C01874=87.153,47.905,41.515,178.9994,1.0610,0.0000
C01875=89.570,44.326,41.678,179.9701,0.0579,0.0000
C01876=91.502,40.323,41.785,179.9964,0.0081,0.0000
C01877=93.214,36.189,41.785,179.9968,0.0083,0.0000
C01878=94.679,31.992,41.678,179.9802,0.0621,0.0000
C01879=95.500,27.752,41.515,179.9573,1.4576,0.0000
C01880=94.968,23.775,41.355,-179.3183,2.1553,0.0000
C01881=93.250,20.743,41.159,-177.2598,2.8295,0.0000
C01882=90.644,19.021,40.789,-176.5682,1.8279,0.0000
C01883=87.735,17.640,40.048,-179.2135,0.3689,0.0000
C01884=85.134,16.299,39.090,175.2426,-2.7030,0.0000
C01885=83.232,14.718,38.165,166.7718,-12.7923,0.0000
C01886=82.260,12.305,37.495,171.8942,-33.8546,0.0000
C01887=82.270,8.324,37.229,-177.9072,-37.5897,0.0000
C01888=82.553,4.208,37.217,-177.5804,-37.7646,0.0000
C01889=82.662,0.000,37.225,179.9996,-37.7945,0.0000
C01890=82.553,-4.208,37.217,177.5810,-37.7647,0.0000
C01891=82.270,-8.324,37.229,177.9089,-37.5895,0.0000
C01892=82.260,-12.305,37.495,-171.8950,-33.8549,0.0000
C01893=83.232,-14.718,38.165,-166.7718,-12.7923,0.0000
C01894=85.134,-16.299,39.090,-175.2426,-2.7030,0.0000
C01895=87.735,-17.640,40.048,179.2135,0.3689,0.0000
C01896=90.644,-19.021,40.789,176.5682,1.8279,0.0000
C01897=93.250,-20.743,41.159,177.2598,2.8295,0.0000
C01898=94.968,-23.775,41.355,179.3183,2.1553,0.0000
C01899=95.500,-27.752,41.515,-179.9573,1.4576,0.0000
C01900=94.679,-31.992,41.678,-179.9802,0.0621,0.0000
C01901=93.214,-36.189,41.785,-179.9968,0.0083,0.0000
C01902=91.502,-40.323,41.785,-179.9964,0.0081,0.0000
C01903=89.570,-44.326,41.678,-179.9701,0.0579,0.0000
C01904=87.153,-47.905,41.515,-178.9994,1.0610,0.0000
C01905=83.964,-50.341,41.355,-177.9940,1.0426,0.0000
C01906=80.606,-51.270,41.159,-176.0647,0.0633,0.0000
C01907=77.545,-50.645,40.789,-176.2827,-1.1365,0.0000
C01908=74.511,-49.565,40.048,-179.1830,-0.2954,0.0000
C01909=71.724,-48.673,39.090,174.7304,1.4587,0.0000
C01910=69.261,-48.447,38.165,161.9042,0.3246,0.0000
C01911=66.868,-49.465,37.495,150.0988,-20.4873,0.0000
C01912=64.059,-52.288,37.229,152.5931,-29.6910,0.0000
C01913=61.349,-55.398,37.217,152.6199,-30.0136,0.0000
C01914=58.451,-58.451,37.225,151.2604,-28.7392,0.0000
C01915=55.398,-61.349,37.217,149.9866,-27.3805,0.0000
C01916=52.288,-64.059,37.229,150.3100,-27.4077,0.0000
C01917=49.465,-66.868,37.495,159.5118,-29.9009,0.0000
C01918=48.447,-69.261,38.165,-179.6754,-18.0958,0.0000
C01919=48.673,-71.724,39.090,-178.5413,-5.2696,0.0000
C01920=49.565,-74.511,40.048,179.7046,0.8170,0.0000
C01921=50.645,-77.545,40.789,178.8635,3.7173,0.0000
C01922=51.270,-80.606,41.159,-179.9367,3.9353,0.0000
C01923=50.341,-83.964,41.355,-178.9574,2.0060,0.0000
C01924=47.905,-87.153,41.515,-178.9390,1.0006,0.0000
C01925=44.326,-89.570,41.678,-179.9421,0.0299,0.0000
C01926=40.323,-91.502,41.785,-179.9919,0.0036,0.0000
C01927=36.189,-93.214,41.785,-179.9917,0.0032,0.0000
C01928=31.992,-94.679,41.678,-179.9379,0.0198,0.0000
C01929=27.752,-95.500,41.515,-178.5424,0.0427,0.0000
C01930=23.775,-94.968,41.355,-177.8447,-0.6817,0.0000
C01931=20.743,-93.250,41.159,-177.1705,-2.7402,0.0000
C01932=19.021,-90.644,40.789,-178.1721,-3.4318,0.0000
C01933=17.640,-87.735,40.048,-179.6311,-0.7865,0.0000
C01934=16.299,-85.134,39.090,177.2970,4.7574,0.0000
C01935=14.718,-83.232,38.165,167.2077,13.2282,0.0000
C01936=12.305,-82.260,37.495,146.1454,8.1058,0.0000
C01937=8.324,-82.270,37.229,142.4103,-2.0928,0.0000
C01938=4.208,-82.553,37.217,142.2354,-2.4196,0.0000
C01939=0.000,-82.662,37.225,142.2055,0.0004,0.0000
C01940=0.000,-82.662,37.225,142.2055,0.0004,0.0000
C01941=-4.208,-82.553,37.217,142.2353,2.4190,0.0000
C01942=-8.324,-82.270,37.229,142.4105,2.0911,0.0000
C01943=-12.305,-82.260,37.495,146.1451,-8.1050,0.0000
C01944=-14.718,-83.232,38.165,167.2077,-13.2282,0.0000
C01945=-16.299,-85.134,39.090,177.2970,-4.7574,0.0000
C01946=-17.640,-87.735,40.048,-179.6311,0.7865,0.0000
C01947=-19.021,-90.644,40.789,-178.1721,3.4318,0.0000
C01948=-20.743,-93.250,41.159,-177.1705,2.7402,0.0000
C01949=-23.775,-94.968,41.355,-177.8447,0.6817,0.0000
C01950=-27.752,-95.500,41.515,-178.5424,-0.0427,0.0000
C01951=-31.992,-94.679,41.678,-179.9379,-0.0198,0.0000
C01952=-36.189,-93.214,41.785,-179.9917,-0.0032,0.0000
C01953=-40.323,-91.502,41.785,-179.9919,-0.0036,0.0000
C01954=-44.326,-89.570,41.678,-179.9421,-0.0299,0.0000
C01955=-47.905,-87.153,41.515,-178.9390,-1.0006,0.0000
C01956=-50.341,-83.964,41.355,-178.9574,-2.0060,0.0000
C01957=-51.270,-80.606,41.159,-179.9367,-3.9353,0.0000
C01958=-50.645,-77.545,40.789,178.8635,-3.7173,0.0000
C01959=-49.565,-74.511,40.048,179.7046,-0.8170,0.0000
C01960=-48.673,-71.724,39.090,-178.5413,5.2696,0.0000
C01961=-48.447,-69.261,38.165,-179.6754,18.0958,0.0000
C01962=-49.465,-66.868,37.495,159.5127,29.9012,0.0000
C01963=-52.288,-64.059,37.229,150.3090,27.4069,0.0000
C01964=-55.398,-61.349,37.217,149.9864,27.3801,0.0000
C01965=-58.451,-58.451,37.225,151.2608,28.7396,0.0000
C01966=-61.349,-55.398,37.217,152.6195,30.0134,0.0000
C01967=-64.059,-52.288,37.229,152.5923,29.6900,0.0000
C01968=-66.868,-49.465,37.495,150.0991,20.4882,0.0000
C01969=-69.261,-48.447,38.165,161.9042,-0.3246,0.0000
C01970=-71.724,-48.673,39.090,174.7304,-1.4587,0.0000
C01971=-74.511,-49.565,40.048,-179.1830,0.2954,0.0000
C01972=-77.545,-50.645,40.789,-176.2827,1.1365,0.0000
C01973=-80.606,-51.270,41.159,-176.0647,-0.0633,0.0000
C01974=-83.964,-50.341,41.355,-177.9940,-1.0426,0.0000
C01975=-87.153,-47.905,41.515,-178.9994,-1.0610,0.0000
C01976=-89.570,-44.326,41.678,-179.9701,-0.0579,0.0000
C01977=-91.502,-40.323,41.785,-179.9964,-0.0081,0.0000
C01978=-93.214,-36.189,41.785,-179.9968,-0.0083,0.0000
C01979=-94.679,-31.992,41.678,-179.9802,-0.0621,0.0000
C01980=-95.500,-27.752,41.515,-179.9573,-1.4576,0.0000
C01981=-94.968,-23.775,41.355,179.3183,-2.1553,0.0000
C01982=-93.250,-20.743,41.159,177.2598,-2.8295,0.0000
C01983=-90.644,-19.021,40.789,176.5682,-1.8279,0.0000
C01984=-87.735,-17.640,40.048,179.2135,-0.3689,0.0000
C01985=-85.134,-16.299,39.090,-175.2426,2.7030,0.0000
C01986=-83.232,-14.718,38.165,-166.7718,12.7923,0.0000
C01987=-82.260,-12.305,37.495,-171.8942,33.8546,0.0000
C01988=-82.270,-8.324,37.229,177.9072,37.5897,0.0000
C01989=-82.553,-4.208,37.217,177.5804,37.7646,0.0000
C01990=-82.662,0.000,37.225,-179.9996,37.7945,0.0000
C01991=-82.553,4.208,37.217,-177.5810,37.7647,0.0000
C01992=-82.270,8.324,37.229,-177.9089,37.5895,0.0000
C01993=-82.260,12.305,37.495,171.8950,33.8549,0.0000
C01994=-83.232,14.718,38.165,166.7718,12.7923,0.0000
C01995=-85.134,16.299,39.090,175.2426,2.7030,0.0000
C01996=-87.735,17.640,40.048,-179.2135,-0.3689,0.0000
C01997=-90.644,19.021,40.789,-176.5682,-1.8279,0.0000
C01998=-93.250,20.743,41.159,-177.2598,-2.8295,0.0000
C01999=-94.968,23.775,41.355,-179.3183,-2.1553,0.0000
///TOOL 0
///POSTYPE ANGLE
///ANGLE
EC00000=-33.2751,0.0000
EC00001=-32.3830,0.0000
EC00002=-31.4965,0.0000
EC00003=-30.3670,0.0000
EC00004=-28.7935,0.0000
EC00005=-26.9678,0.0000
EC00006=-25.1253,0.0000
EC00007=-23.3660,0.0000
EC00008=-21.6343,0.0000
EC00009=-19.8748,0.0000
EC00010=-18.0324,0.0000
EC00011=-16.2063,0.0000
EC00012=-14.6333,0.0000
EC00013=-13.5035,0.0000
EC00014=-12.6169,0.0000
EC00015=-11.7253,0.0000
EC00016=-10.5819,0.0000
EC00017=-8.8371,0.0000
EC00018=-6.1699,0.0000
EC00019=-3.2152,0.0000
EC00020=0.0000,0.0000
EC00021=0.0000,0.0000
EC00022=3.1930,0.0000
EC00023=6.1402,0.0000
EC00024=8.8129,0.0000
EC00025=10.5402,0.0000
EC00026=11.6582,0.0000
EC00027=12.5225,0.0000
EC00028=13.3766,0.0000
EC00029=14.4702,0.0000
EC00030=16.0363,0.0000
EC00031=17.8866,0.0000
EC00032=19.7782,0.0000
EC00033=21.6011,0.0000
EC00034=23.3991,0.0000
EC00035=25.2213,0.0000
EC00036=27.1138,0.0000
EC00037=28.9637,0.0000
EC00038=30.5297,0.0000
EC00039=31.6234,0.0000
EC00040=32.4779,0.0000
EC00041=33.3415,0.0000
EC00042=34.4600,0.0000
EC00043=36.1873,0.0000
EC00044=38.8598,0.0000
EC00045=41.8071,0.0000
EC00046=45.0000,0.0000
EC00047=48.1929,0.0000
EC00048=51.1402,0.0000
EC00049=53.8127,0.0000
EC00050=55.5400,0.0000
EC00051=56.6585,0.0000
EC00052=57.5221,0.0000
EC00053=58.3766,0.0000
EC00054=59.4703,0.0000
EC00055=61.0363,0.0000
EC00056=62.8862,0.0000
EC00057=64.7787,0.0000
EC00058=66.6009,0.0000
EC00059=68.3989,0.0000
EC00060=70.2218,0.0000
EC00061=72.1134,0.0000
EC00062=73.9637,0.0000
EC00063=75.5298,0.0000
EC00064=76.6234,0.0000
EC00065=77.4775,0.0000
EC00066=78.3418,0.0000
EC00067=79.4598,0.0000
EC00068=81.1871,0.0000
EC00069=83.8598,0.0000
EC00070=86.8070,0.0000
EC00071=90.0000,0.0000
EC00072=93.1930,0.0000
EC00073=96.1402,0.0000
EC00074=98.8128,0.0000
EC00075=100.5402,0.0000
EC00076=101.6582,0.0000
EC00077=102.5225,0.0000
EC00078=103.3766,0.0000
EC00079=104.4702,0.0000
EC00080=106.0363,0.0000
EC00081=107.8866,0.0000
EC00082=109.7782,0.0000
EC00083=111.6011,0.0000
EC00084=113.3991,0.0000
EC00085=115.2213,0.0000
EC00086=117.1138,0.0000
EC00087=118.9637,0.0000
EC00088=120.5297,0.0000
EC00089=121.6234,0.0000
EC00090=122.4779,0.0000
EC00091=123.3415,0.0000
EC00092=124.4600,0.0000
EC00093=126.1873,0.0000
EC00094=128.8598,0.0000
EC00095=131.8071,0.0000
EC00096=135.0000,0.0000
EC00097=138.1929,0.0000
EC00098=141.1402,0.0000
EC00099=143.8127,0.0000
EC00100=145.5400,0.0000
EC00101=146.6585,0.0000
EC00102=147.5221,0.0000
EC00103=148.3766,0.0000
EC00104=149.4703,0.0000
EC00105=151.0363,0.0000
EC00106=152.8862,0.0000
EC00107=154.7787,0.0000
EC00108=156.6009,0.0000
EC00109=158.3989,0.0000
EC00110=160.2218,0.0000
EC00111=162.1134,0.0000
EC00112=163.9637,0.0000
EC00113=165.5298,0.0000
EC00114=166.6234,0.0000
EC00115=167.4775,0.0000
EC00116=168.3418,0.0000
EC00117=169.4598,0.0000
EC00118=171.1871,0.0000
EC00119=173.8598,0.0000
EC00120=176.8070,0.0000
EC00121=180.0000,0.0000
EC00122=180.0000,0.0000
EC00123=-176.8070,0.0000
EC00124=-173.8598,0.0000
EC00125=-171.1872,0.0000
EC00126=-169.4598,0.0000
EC00127=-168.3418,0.0000
EC00128=-167.4775,0.0000
EC00129=-166.6234,0.0000
EC00130=-165.5298,0.0000
EC00131=-163.9637,0.0000
EC00132=-162.1134,0.0000
EC00133=-160.2218,0.0000
EC00134=-158.3989,0.0000
EC00135=-156.6009,0.0000
EC00136=-154.7787,0.0000
EC00137=-152.8862,0.0000
EC00138=-151.0363,0.0000
EC00139=-149.4703,0.0000
EC00140=-148.3766,0.0000
EC00141=-147.5221,0.0000
EC00142=-146.6585,0.0000
EC00143=-145.5400,0.0000
EC00144=-143.8127,0.0000
EC00145=-141.1402,0.0000
EC00146=-138.1929,0.0000
EC00147=-135.0000,0.0000
EC00148=-131.8071,0.0000
EC00149=-128.8598,0.0000
EC00150=-126.1873,0.0000
EC00151=-124.4600,0.0000
EC00152=-123.3415,0.0000
EC00153=-122.4779,0.0000
EC00154=-121.6234,0.0000
EC00155=-120.5297,0.0000
EC00156=-118.9637,0.0000
EC00157=-117.1138,0.0000
EC00158=-115.2213,0.0000
EC00159=-113.3991,0.0000
EC00160=-111.6011,0.0000
EC00161=-109.7782,0.0000
EC00162=-107.8866,0.0000
EC00163=-106.0363,0.0000
EC00164=-104.4702,0.0000
EC00165=-103.3766,0.0000
EC00166=-102.5225,0.0000
EC00167=-101.6582,0.0000
EC00168=-100.5402,0.0000
EC00169=-98.8129,0.0000
EC00170=-96.1402,0.0000
EC00171=-93.1930,0.0000
EC00172=-90.0000,0.0000
EC00173=-86.8070,0.0000
EC00174=-83.8598,0.0000
EC00175=-81.1872,0.0000
EC00176=-79.4598,0.0000
EC00177=-78.3418,0.0000
EC00178=-77.4775,0.0000
EC00179=-76.6234,0.0000
EC00180=-75.5298,0.0000
EC00181=-73.9637,0.0000
EC00182=-72.1134,0.0000
EC00183=-70.2218,0.0000
EC00184=-68.3989,0.0000
EC00185=-66.6009,0.0000
EC00186=-64.7787,0.0000
EC00187=-62.8862,0.0000
EC00188=-61.0363,0.0000
EC00189=-59.4703,0.0000
EC00190=-58.3766,0.0000
EC00191=-57.5221,0.0000
EC00192=-56.6585,0.0000
EC00193=-55.5400,0.0000
EC00194=-53.8127,0.0000
EC00195=-51.1402,0.0000
EC00196=-48.1929,0.0000
EC00197=-45.0000,0.0000
EC00198=-41.8071,0.0000
EC00199=-38.8598,0.0000
EC00200=-36.1873,0.0000
EC00201=-34.4600,0.0000
EC00202=-33.3415,0.0000
EC00203=-32.4779,0.0000
EC00204=-31.6234,0.0000
EC00205=-30.5297,0.0000
EC00206=-28.9637,0.0000
EC00207=-27.1138,0.0000
EC00208=-25.2213,0.0000
EC00209=-23.3991,0.0000
EC00210=-21.6011,0.0000
EC00211=-19.7782,0.0000
EC00212=-17.8866,0.0000
EC00213=-16.0363,0.0000
EC00214=-14.4702,0.0000
EC00215=-13.3766,0.0000
EC00216=-12.5225,0.0000
EC00217=-11.6582,0.0000
EC00218=-10.5402,0.0000
EC00219=-8.8128,0.0000
EC00220=-6.1402,0.0000
EC00221=-3.1930,0.0000
EC00222=0.0000,0.0000
EC00223=0.0000,0.0000
EC00224=3.1693,0.0000
EC00225=6.1086,0.0000
EC00226=8.7858,0.0000
EC00227=10.4951,0.0000
EC00228=11.5862,0.0000
EC00229=12.4199,0.0000
EC00230=13.2394,0.0000
EC00231=14.2944,0.0000
EC00232=15.8535,0.0000
EC00233=17.7299,0.0000
EC00234=19.6757,0.0000
EC00235=21.5655,0.0000
EC00236=23.4348,0.0000
EC00237=25.3246,0.0000
EC00238=27.2701,0.0000
EC00239=29.1464,0.0000
EC00240=30.7059,0.0000
EC00241=31.7605,0.0000
EC00242=32.5800,0.0000
EC00243=33.4139,0.0000
EC00244=34.5045,0.0000
EC00245=36.2144,0.0000
EC00246=38.8913,0.0000
EC00247=41.8309,0.0000
EC00248=45.0000,0.0000
EC00249=48.1691,0.0000
EC00250=51.1087,0.0000
EC00251=53.7856,0.0000
EC00252=55.4955,0.0000
EC00253=56.5861,0.0000
EC00254=57.4200,0.0000
EC00255=58.2395,0.0000
EC00256=59.2941,0.0000
EC00257=60.8536,0.0000
EC00258=62.7299,0.0000
EC00259=64.6754,0.0000
EC00260=66.5652,0.0000
EC00261=68.4345,0.0000
EC00262=70.3243,0.0000
EC00263=72.2701,0.0000
EC00264=74.1465,0.0000
EC00265=75.7056,0.0000
EC00266=76.7606,0.0000
EC00267=77.5801,0.0000
EC00268=78.4138,0.0000
EC00269=79.5049,0.0000
EC00270=81.2142,0.0000
EC00271=83.8914,0.0000
EC00272=86.8307,0.0000
EC00273=90.0000,0.0000
EC00274=93.1693,0.0000
EC00275=96.1086,0.0000
EC00276=98.7858,0.0000
EC00277=100.4951,0.0000
EC00278=101.5862,0.0000
EC00279=102.4199,0.0000
EC00280=103.2394,0.0000
EC00281=104.2944,0.0000
EC00282=105.8535,0.0000
EC00283=107.7299,0.0000
EC00284=109.6757,0.0000
EC00285=111.5655,0.0000
EC00286=113.4348,0.0000
EC00287=115.3246,0.0000
EC00288=117.2701,0.0000
EC00289=119.1464,0.0000
EC00290=120.7059,0.0000
EC00291=121.7605,0.0000
EC00292=122.5800,0.0000
EC00293=123.4139,0.0000
EC00294=124.5045,0.0000
EC00295=126.2144,0.0000
EC00296=128.8913,0.0000
EC00297=131.8309,0.0000
EC00298=135.0000,0.0000
EC00299=138.1691,0.0000
EC00300=141.1087,0.0000
EC00301=143.7856,0.0000
EC00302=145.4955,0.0000
EC00303=146.5861,0.0000
EC00304=147.4200,0.0000
EC00305=148.2395,0.0000
EC00306=149.2941,0.0000
EC00307=150.8536,0.0000
EC00308=152.7299,0.0000
EC00309=154.6754,0.0000
EC00310=156.5652,0.0000
EC00311=158.4345,0.0000
EC00312=160.3243,0.0000
EC00313=162.2701,0.0000
EC00314=164.1465,0.0000
EC00315=165.7056,0.0000
EC00316=166.7606,0.0000
EC00317=167.5801,0.0000
EC00318=168.4138,0.0000
EC00319=169.5049,0.0000
EC00320=171.2142,0.0000
EC00321=173.8914,0.0000
EC00322=176.8307,0.0000
EC00323=180.0000,0.0000
EC00324=180.0000,0.0000
EC00325=-176.8307,0.0000
EC00326=-173.8914,0.0000
EC00327=-171.2142,0.0000
EC00328=-169.5049,0.0000
EC00329=-168.4138,0.0000
EC00330=-167.5801,0.0000
EC00331=-166.7606,0.0000
EC00332=-165.7056,0.0000
EC00333=-164.1465,0.0000
EC00334=-162.2701,0.0000
EC00335=-160.3243,0.0000
EC00336=-158.4345,0.0000
EC00337=-156.5652,0.0000
EC00338=-154.6754,0.0000
EC00339=-152.7299,0.0000
EC00340=-150.8536,0.0000
EC00341=-149.2941,0.0000
EC00342=-148.2395,0.0000
EC00343=-147.4200,0.0000
EC00344=-146.5861,0.0000
EC00345=-145.4955,0.0000
EC00346=-143.7856,0.0000
EC00347=-141.1087,0.0000
EC00348=-138.1691,0.0000
EC00349=-135.0000,0.0000
EC00350=-131.8309,0.0000
EC00351=-128.8913,0.0000
EC00352=-126.2144,0.0000
EC00353=-124.5045,0.0000
EC00354=-123.4139,0.0000
EC00355=-122.5800,0.0000
EC00356=-121.7605,0.0000
EC00357=-120.7059,0.0000
EC00358=-119.1464,0.0000
EC00359=-117.2701,0.0000
EC00360=-115.3246,0.0000
EC00361=-113.4348,0.0000
EC00362=-111.5655,0.0000
EC00363=-109.6757,0.0000
EC00364=-107.7299,0.0000
EC00365=-105.8535,0.0000
EC00366=-104.2944,0.0000
EC00367=-103.2394,0.0000
EC00368=-102.4199,0.0000
EC00369=-101.5862,0.0000
EC00370=-100.4951,0.0000
EC00371=-98.7858,0.0000
EC00372=-96.1086,0.0000
EC00373=-93.1693,0.0000
EC00374=-90.0000,0.0000
EC00375=-86.8307,0.0000
EC00376=-83.8914,0.0000
EC00377=-81.2142,0.0000
EC00378=-79.5049,0.0000
EC00379=-78.4138,0.0000
EC00380=-77.5801,0.0000
EC00381=-76.7606,0.0000
EC00382=-75.7056,0.0000
EC00383=-74.1465,0.0000
EC00384=-72.2701,0.0000
EC00385=-70.3243,0.0000
EC00386=-68.4345,0.0000
EC00387=-66.5652,0.0000
EC00388=-64.6754,0.0000
EC00389=-62.7299,0.0000
EC00390=-60.8536,0.0000
EC00391=-59.2941,0.0000
EC00392=-58.2395,0.0000
EC00393=-57.4200,0.0000
EC00394=-56.5861,0.0000
EC00395=-55.4955,0.0000
EC00396=-53.7856,0.0000
EC00397=-51.1087,0.0000
EC00398=-48.1691,0.0000
EC00399=-45.0000,0.0000
EC00400=-41.8309,0.0000
EC00401=-38.8913,0.0000
EC00402=-36.2144,0.0000
EC00403=-34.5045,0.0000
EC00404=-33.4139,0.0000
EC00405=-32.5800,0.0000
EC00406=-31.7605,0.0000
EC00407=-30.7059,0.0000
EC00408=-29.1464,0.0000
EC00409=-27.2701,0.0000
EC00410=-25.3246,0.0000
EC00411=-23.4348,0.0000
EC00412=-21.5655,0.0000
EC00413=-19.6757,0.0000
EC00414=-17.7299,0.0000
EC00415=-15.8535,0.0000
EC00416=-14.2944,0.0000
EC00417=-13.2394,0.0000
EC00418=-12.4199,0.0000
EC00419=-11.5862,0.0000
EC00420=-10.4951,0.0000
EC00421=-8.7858,0.0000
EC00422=-6.1086,0.0000
EC00423=-3.1693,0.0000
EC00424=0.0000,0.0000
EC00425=0.0000,0.0000
EC00426=3.1434,0.0000
EC00427=6.0750,0.0000
EC00428=8.7577,0.0000
EC00429=10.4474,0.0000
EC00430=11.5089,0.0000
EC00431=12.3101,0.0000
EC00432=13.0930,0.0000
EC00433=14.1066,0.0000
EC00434=15.6587,0.0000
EC00435=17.5637,0.0000
EC00436=19.5659,0.0000
EC00437=21.5274,0.0000
EC00438=23.4725,0.0000
EC00439=25.4343,0.0000
EC00440=27.4359,0.0000
EC00441=29.3411,0.0000
EC00442=30.8935,0.0000
EC00443=31.9071,0.0000
EC00444=32.6899,0.0000
EC00445=33.4910,0.0000
EC00446=34.5530,0.0000
EC00447=36.2423,0.0000
EC00448=38.9252,0.0000
EC00449=41.8567,0.0000
EC00450=45.0000,0.0000
EC00451=48.1433,0.0000
EC00452=51.0748,0.0000
EC00453=53.7577,0.0000
EC00454=55.4470,0.0000
EC00455=56.5090,0.0000
EC00456=57.3101,0.0000
EC00457=58.0929,0.0000
EC00458=59.1065,0.0000
EC00459=60.6589,0.0000
EC00460=62.5641,0.0000
EC00461=64.5657,0.0000
EC00462=66.5275,0.0000
EC00463=68.4726,0.0000
EC00464=70.4341,0.0000
EC00465=72.4363,0.0000
EC00466=74.3413,0.0000
EC00467=75.8934,0.0000
EC00468=76.9070,0.0000
EC00469=77.6899,0.0000
EC00470=78.4911,0.0000
EC00471=79.5526,0.0000
EC00472=81.2423,0.0000
EC00473=83.9250,0.0000
EC00474=86.8566,0.0000
EC00475=90.0000,0.0000
EC00476=93.1434,0.0000
EC00477=96.0750,0.0000
EC00478=98.7577,0.0000
EC00479=100.4474,0.0000
EC00480=101.5089,0.0000
EC00481=102.3101,0.0000
EC00482=103.0930,0.0000
EC00483=104.1066,0.0000
EC00484=105.6587,0.0000
EC00485=107.5637,0.0000
EC00486=109.5659,0.0000
EC00487=111.5274,0.0000
EC00488=113.4725,0.0000
EC00489=115.4343,0.0000
EC00490=117.4359,0.0000
EC00491=119.3411,0.0000
EC00492=120.8935,0.0000
EC00493=121.9071,0.0000
EC00494=122.6899,0.0000
EC00495=123.4910,0.0000
EC00496=124.5530,0.0000
EC00497=126.2423,0.0000
EC00498=128.9252,0.0000
EC00499=131.8567,0.0000
EC00500=135.0000,0.0000
EC00501=138.1433,0.0000
EC00502=141.0748,0.0000
EC00503=143.7577,0.0000
EC00504=145.4470,0.0000
EC00505=146.5090,0.0000
EC00506=147.3101,0.0000
EC00507=148.0929,0.0000
EC00508=149.1065,0.0000
EC00509=150.6589,0.0000
EC00510=152.5641,0.0000
EC00511=154.5657,0.0000
EC00512=156.5275,0.0000
EC00513=158.4726,0.0000
EC00514=160.4341,0.0000
EC00515=162.4363,0.0000
EC00516=164.3413,0.0000
EC00517=165.8934,0.0000
EC00518=166.9070,0.0000
EC00519=167.6899,0.0000
EC00520=168.4911,0.0000
EC00521=169.5526,0.0000
EC00522=171.2423,0.0000
EC00523=173.9250,0.0000
EC00524=176.8566,0.0000
EC00525=180.0000,0.0000
EC00526=180.0000,0.0000
EC00527=-176.8566,0.0000
EC00528=-173.9250,0.0000
EC00529=-171.2423,0.0000
EC00530=-169.5526,0.0000
EC00531=-168.4911,0.0000
EC00532=-167.6899,0.0000
EC00533=-166.9070,0.0000
EC00534=-165.8934,0.0000
EC00535=-164.3413,0.0000
EC00536=-162.4363,0.0000
EC00537=-160.4341,0.0000
EC00538=-158.4726,0.0000
EC00539=-156.5275,0.0000
EC00540=-154.5657,0.0000
EC00541=-152.5641,0.0000
EC00542=-150.6589,0.0000
EC00543=-149.1065,0.0000
EC00544=-148.0929,0.0000
EC00545=-147.3101,0.0000
EC00546=-146.5090,0.0000
EC00547=-145.4470,0.0000
EC00548=-143.7577,0.0000
EC00549=-141.0748,0.0000
EC00550=-138.1433,0.0000
EC00551=-135.0000,0.0000
EC00552=-131.8567,0.0000
EC00553=-128.9252,0.0000
EC00554=-126.2423,0.0000
EC00555=-124.5530,0.0000
EC00556=-123.4910,0.0000
EC00557=-122.6899,0.0000
EC00558=-121.9071,0.0000
EC00559=-120.8935,0.0000
EC00560=-119.3411,0.0000
EC00561=-117.4359,0.0000
EC00562=-115.4343,0.0000
EC00563=-113.4725,0.0000
EC00564=-111.5274,0.0000
EC00565=-109.5659,0.0000
EC00566=-107.5637,0.0000
EC00567=-105.6587,0.0000
EC00568=-104.1066,0.0000
EC00569=-103.0930,0.0000
EC00570=-102.3101,0.0000
EC00571=-101.5089,0.0000
EC00572=-100.4474,0.0000
EC00573=-98.7577,0.0000
EC00574=-96.0750,0.0000
EC00575=-93.1434,0.0000
EC00576=-90.0000,0.0000
EC00577=-86.8566,0.0000
EC00578=-83.9250,0.0000
EC00579=-81.2423,0.0000
EC00580=-79.5526,0.0000
EC00581=-78.4911,0.0000
EC00582=-77.6899,0.0000
EC00583=-76.9070,0.0000
EC00584=-75.8934,0.0000
EC00585=-74.3413,0.0000
EC00586=-72.4363,0.0000
EC00587=-70.4341,0.0000
EC00588=-68.4726,0.0000
EC00589=-66.5275,0.0000
EC00590=-64.5657,0.0000
EC00591=-62.5641,0.0000
EC00592=-60.6589,0.0000
EC00593=-59.1065,0.0000
EC00594=-58.0929,0.0000
EC00595=-57.3101,0.0000
EC00596=-56.5090,0.0000
EC00597=-55.4470,0.0000
EC00598=-53.7577,0.0000
EC00599=-51.0748,0.0000
EC00600=-48.1433,0.0000
EC00601=-45.0000,0.0000
EC00602=-41.8567,0.0000
EC00603=-38.9252,0.0000
EC00604=-36.2423,0.0000
EC00605=-34.5530,0.0000
EC00606=-33.4910,0.0000
EC00607=-32.6899,0.0000
EC00608=-31.9071,0.0000
EC00609=-30.8935,0.0000
EC00610=-29.3411,0.0000
EC00611=-27.4359,0.0000
EC00612=-25.4343,0.0000
EC00613=-23.4725,0.0000
EC00614=-21.5274,0.0000
EC00615=-19.5659,0.0000
EC00616=-17.5637,0.0000
EC00617=-15.6587,0.0000
EC00618=-14.1066,0.0000
EC00619=-13.0930,0.0000
EC00620=-12.3101,0.0000
EC00621=-11.5089,0.0000
EC00622=-10.4474,0.0000
EC00623=-8.7577,0.0000
EC00624=-6.0750,0.0000
EC00625=-3.1434,0.0000
EC00626=0.0000,0.0000
EC00627=0.0000,0.0000
EC00628=3.1159,0.0000
EC00629=6.0385,0.0000
EC00630=8.7274,0.0000
EC00631=10.3963,0.0000
EC00632=11.4267,0.0000
EC00633=12.1938,0.0000
EC00634=12.9380,0.0000
EC00635=13.9087,0.0000
EC00636=15.4538,0.0000
EC00637=17.3887,0.0000
EC00638=19.4506,0.0000
EC00639=21.4875,0.0000
EC00640=23.5125,0.0000
EC00641=25.5494,0.0000
EC00642=27.6113,0.0000
EC00643=29.5463,0.0000
EC00644=31.0916,0.0000
EC00645=32.0621,0.0000
EC00646=32.8061,0.0000
EC00647=33.5730,0.0000
EC00648=34.6038,0.0000
EC00649=36.2732,0.0000
EC00650=38.9613,0.0000
EC00651=41.8843,0.0000
EC00652=45.0000,0.0000
EC00653=48.1157,0.0000
EC00654=51.0387,0.0000
EC00655=53.7268,0.0000
EC00656=55.3962,0.0000
EC00657=56.4270,0.0000
EC00658=57.1939,0.0000
EC00659=57.9379,0.0000
EC00660=58.9084,0.0000
EC00661=60.4537,0.0000
EC00662=62.3887,0.0000
EC00663=64.4506,0.0000
EC00664=66.4875,0.0000
EC00665=68.5125,0.0000
EC00666=70.5494,0.0000
EC00667=72.6113,0.0000
EC00668=74.5462,0.0000
EC00669=76.0913,0.0000
EC00670=77.0620,0.0000
EC00671=77.8062,0.0000
EC00672=78.5733,0.0000
EC00673=79.6037,0.0000
EC00674=81.2726,0.0000
EC00675=83.9615,0.0000
EC00676=86.8841,0.0000
EC00677=90.0000,0.0000
EC00678=93.1159,0.0000
EC00679=96.0385,0.0000
EC00680=98.7274,0.0000
EC00681=100.3963,0.0000
EC00682=101.4267,0.0000
EC00683=102.1938,0.0000
EC00684=102.9380,0.0000
EC00685=103.9087,0.0000
EC00686=105.4538,0.0000
EC00687=107.3887,0.0000
EC00688=109.4506,0.0000
EC00689=111.4875,0.0000
EC00690=113.5125,0.0000
EC00691=115.5494,0.0000
EC00692=117.6113,0.0000
EC00693=119.5463,0.0000
EC00694=121.0916,0.0000
EC00695=122.0621,0.0000
EC00696=122.8061,0.0000
EC00697=123.5730,0.0000
EC00698=124.6038,0.0000
EC00699=126.2732,0.0000
EC00700=128.9613,0.0000
EC00701=131.8843,0.0000
EC00702=135.0000,0.0000
EC00703=138.1157,0.0000
EC00704=141.0387,0.0000
EC00705=143.7268,0.0000
EC00706=145.3962,0.0000
EC00707=146.4270,0.0000
EC00708=147.1939,0.0000
EC00709=147.9379,0.0000
EC00710=148.9084,0.0000
EC00711=150.4537,0.0000
EC00712=152.3887,0.0000
EC00713=154.4506,0.0000
EC00714=156.4875,0.0000
EC00715=158.5125,0.0000
EC00716=160.5494,0.0000
EC00717=162.6113,0.0000
EC00718=164.5462,0.0000
EC00719=166.0913,0.0000
EC00720=167.0620,0.0000
EC00721=167.8062,0.0000
EC00722=168.5733,0.0000
EC00723=169.6037,0.0000
EC00724=171.2726,0.0000
EC00725=173.9615,0.0000
EC00726=176.8841,0.0000
EC00727=180.0000,0.0000
EC00728=180.0000,0.0000
EC00729=-176.8841,0.0000
EC00730=-173.9615,0.0000
EC00731=-171.2726,0.0000
EC00732=-169.6037,0.0000
EC00733=-168.5733,0.0000
EC00734=-167.8062,0.0000
EC00735=-167.0620,0.0000
EC00736=-166.0913,0.0000
EC00737=-164.5462,0.0000
EC00738=-162.6113,0.0000
EC00739=-160.5494,0.0000
EC00740=-158.5125,0.0000
EC00741=-156.4875,0.0000
EC00742=-154.4506,0.0000
EC00743=-152.3887,0.0000
EC00744=-150.4537,0.0000
EC00745=-148.9084,0.0000
EC00746=-147.9379,0.0000
EC00747=-147.1939,0.0000
EC00748=-146.4270,0.0000
EC00749=-145.3962,0.0000
EC00750=-143.7268,0.0000
EC00751=-141.0387,0.0000
EC00752=-138.1157,0.0000
EC00753=-135.0000,0.0000
EC00754=-131.8843,0.0000
EC00755=-128.9613,0.0000
EC00756=-126.2732,0.0000
EC00757=-124.6038,0.0000
EC00758=-123.5730,0.0000
EC00759=-122.8061,0.0000
EC00760=-122.0621,0.0000
EC00761=-121.0916,0.0000
EC00762=-119.5463,0.0000
EC00763=-117.6113,0.0000
EC00764=-115.5494,0.0000
EC00765=-113.5125,0.0000
EC00766=-111.4875,0.0000
EC00767=-109.4506,0.0000
EC00768=-107.3887,0.0000
EC00769=-105.4538,0.0000
EC00770=-103.9087,0.0000
EC00771=-102.9380,0.0000
EC00772=-102.1938,0.0000
EC00773=-101.4267,0.0000
EC00774=-100.3963,0.0000
EC00775=-98.7274,0.0000
EC00776=-96.0385,0.0000
EC00777=-93.1159,0.0000
EC00778=-90.0000,0.0000
EC00779=-86.8841,0.0000
EC00780=-83.9615,0.0000
EC00781=-81.2726,0.0000
EC00782=-79.6037,0.0000
EC00783=-78.5733,0.0000
EC00784=-77.8062,0.0000
EC00785=-77.0620,0.0000
EC00786=-76.0913,0.0000
EC00787=-74.5462,0.0000
EC00788=-72.6113,0.0000
EC00789=-70.5494,0.0000
EC00790=-68.5125,0.0000
EC00791=-66.4875,0.0000
EC00792=-64.4506,0.0000
EC00793=-62.3887,0.0000
EC00794=-60.4537,0.0000
EC00795=-58.9084,0.0000
EC00796=-57.9379,0.0000
EC00797=-57.1939,0.0000
EC00798=-56.4270,0.0000
EC00799=-55.3962,0.0000
EC00800=-53.7268,0.0000
EC00801=-51.0387,0.0000
EC00802=-48.1157,0.0000
EC00803=-45.0000,0.0000
EC00804=-41.8843,0.0000
EC00805=-38.9613,0.0000
EC00806=-36.2732,0.0000
EC00807=-34.6038,0.0000
EC00808=-33.5730,0.0000
EC00809=-32.8061,0.0000
EC00810=-32.0621,0.0000
EC00811=-31.0916,0.0000
EC00812=-29.5463,0.0000
EC00813=-27.6113,0.0000
EC00814=-25.5494,0.0000
EC00815=-23.5125,0.0000
EC00816=-21.4875,0.0000
EC00817=-19.4506,0.0000
EC00818=-17.3887,0.0000
EC00819=-15.4538,0.0000
EC00820=-13.9087,0.0000
EC00821=-12.9380,0.0000
EC00822=-12.1938,0.0000
EC00823=-11.4267,0.0000
EC00824=-10.3963,0.0000
EC00825=-8.7274,0.0000
EC00826=-6.0385,0.0000
EC00827=-3.1159,0.0000
EC00828=0.0000,0.0000
EC00829=0.0000,0.0000
EC00830=3.0871,0.0000
EC00831=6.0002,0.0000
EC00832=8.6952,0.0000
EC00833=10.3419,0.0000
EC00834=11.3400,0.0000
EC00835=12.0705,0.0000
EC00836=12.7745,0.0000
EC00837=13.7009,0.0000
EC00838=15.2391,0.0000
EC00839=17.2060,0.0000
EC00840=19.3299,0.0000
EC00841=21.4458,0.0000
EC00842=23.5540,0.0000
EC00843=25.6698,0.0000
EC00844=27.7938,0.0000
EC00845=29.7609,0.0000
EC00846=31.2994,0.0000
EC00847=32.2255,0.0000
EC00848=32.9290,0.0000
EC00849=33.6599,0.0000
EC00850=34.6583,0.0000
EC00851=36.3048,0.0000
EC00852=38.9993,0.0000
EC00853=41.9128,0.0000
EC00854=45.0000,0.0000
EC00855=48.0872,0.0000
EC00856=51.0007,0.0000
EC00857=53.6952,0.0000
EC00858=55.3417,0.0000
EC00859=56.3401,0.0000
EC00860=57.0710,0.0000
EC00861=57.7745,0.0000
EC00862=58.7006,0.0000
EC00863=60.2391,0.0000
EC00864=62.2062,0.0000
EC00865=64.3302,0.0000
EC00866=66.4460,0.0000
EC00867=68.5542,0.0000
EC00868=70.6701,0.0000
EC00869=72.7940,0.0000
EC00870=74.7609,0.0000
EC00871=76.2991,0.0000
EC00872=77.2255,0.0000
EC00873=77.9295,0.0000
EC00874=78.6600,0.0000
EC00875=79.6581,0.0000
EC00876=81.3048,0.0000
EC00877=83.9998,0.0000
EC00878=86.9129,0.0000
EC00879=90.0000,0.0000
EC00880=93.0871,0.0000
EC00881=96.0002,0.0000
EC00882=98.6952,0.0000
EC00883=100.3419,0.0000
EC00884=101.3400,0.0000
EC00885=102.0705,0.0000
EC00886=102.7745,0.0000
EC00887=103.7009,0.0000
EC00888=105.2391,0.0000
EC00889=107.2060,0.0000
EC00890=109.3299,0.0000
EC00891=111.4458,0.0000
EC00892=113.5540,0.0000
EC00893=115.6698,0.0000
EC00894=117.7938,0.0000
EC00895=119.7609,0.0000
EC00896=121.2994,0.0000
EC00897=122.2255,0.0000
EC00898=122.9290,0.0000
EC00899=123.6599,0.0000
EC00900=124.6583,0.0000
EC00901=126.3048,0.0000
EC00902=128.9993,0.0000
EC00903=131.9128,0.0000
EC00904=135.0000,0.0000
EC00905=138.0872,0.0000
EC00906=141.0007,0.0000
EC00907=143.6952,0.0000
EC00908=145.3417,0.0000
EC00909=146.3401,0.0000
EC00910=147.0710,0.0000
EC00911=147.7745,0.0000
EC00912=148.7006,0.0000
EC00913=150.2391,0.0000
EC00914=152.2062,0.0000
EC00915=154.3302,0.0000
EC00916=156.4460,0.0000
EC00917=158.5542,0.0000
EC00918=160.6701,0.0000
EC00919=162.7940,0.0000
EC00920=164.7609,0.0000
EC00921=166.2991,0.0000
EC00922=167.2255,0.0000
EC00923=167.9295,0.0000
EC00924=168.6600,0.0000
EC00925=169.6581,0.0000
EC00926=171.3048,0.0000
EC00927=173.9998,0.0000
EC00928=176.9129,0.0000
EC00929=180.0000,0.0000
EC00930=180.0000,0.0000
EC00931=-176.9129,0.0000
EC00932=-173.9998,0.0000
EC00933=-171.3048,0.0000
EC00934=-169.6581,0.0000
EC00935=-168.6600,0.0000
EC00936=-167.9295,0.0000
EC00937=-167.2255,0.0000
EC00938=-166.2991,0.0000
EC00939=-164.7609,0.0000
EC00940=-162.7940,0.0000
EC00941=-160.6701,0.0000
EC00942=-158.5542,0.0000
EC00943=-156.4460,0.0000
EC00944=-154.3302,0.0000
EC00945=-152.2062,0.0000
EC00946=-150.2391,0.0000
EC00947=-148.7006,0.0000
EC00948=-147.7745,0.0000
EC00949=-147.0710,0.0000
EC00950=-146.3401,0.0000
EC00951=-145.3417,0.0000
EC00952=-143.6952,0.0000
EC00953=-141.0007,0.0000
EC00954=-138.0872,0.0000
EC00955=-135.0000,0.0000
EC00956=-131.9128,0.0000
EC00957=-128.9993,0.0000
EC00958=-126.3048,0.0000
EC00959=-124.6583,0.0000
EC00960=-123.6599,0.0000
EC00961=-122.9290,0.0000
EC00962=-122.2255,0.0000
EC00963=-121.2994,0.0000
EC00964=-119.7609,0.0000
EC00965=-117.7938,0.0000
EC00966=-115.6698,0.0000
EC00967=-113.5540,0.0000
EC00968=-111.4458,0.0000
EC00969=-109.3299,0.0000
EC00970=-107.2060,0.0000
EC00971=-105.2391,0.0000
EC00972=-103.7009,0.0000
EC00973=-102.7745,0.0000
EC00974=-102.0705,0.0000
EC00975=-101.3400,0.0000
EC00976=-100.3419,0.0000
EC00977=-98.6952,0.0000
EC00978=-96.0002,0.0000
EC00979=-93.0871,0.0000
EC00980=-90.0000,0.0000
EC00981=-86.9129,0.0000
EC00982=-83.9998,0.0000
EC00983=-81.3048,0.0000
EC00984=-79.6581,0.0000
EC00985=-78.6600,0.0000
EC00986=-77.9295,0.0000
EC00987=-77.2255,0.0000
EC00988=-76.2991,0.0000
EC00989=-74.7609,0.0000
EC00990=-72.7940,0.0000
EC00991=-70.6701,0.0000
EC00992=-68.5542,0.0000
EC00993=-66.4460,0.0000
EC00994=-64.3302,0.0000
EC00995=-62.2062,0.0000
EC00996=-60.2391,0.0000
EC00997=-58.7006,0.0000
EC00998=-57.7745,0.0000
EC00999=-57.0710,0.0000
EC01000=-56.3401,0.0000
EC01001=-55.3417,0.0000
EC01002=-53.6952,0.0000
EC01003=-51.0007,0.0000
EC01004=-48.0872,0.0000
EC01005=-45.0000,0.0000
EC01006=-41.9128,0.0000
EC01007=-38.9993,0.0000
EC01008=-36.3048,0.0000
EC01009=-34.6583,0.0000
EC01010=-33.6599,0.0000
EC01011=-32.9290,0.0000
EC01012=-32.2255,0.0000
EC01013=-31.2994,0.0000
EC01014=-29.7609,0.0000
EC01015=-27.7938,0.0000
EC01016=-25.6698,0.0000
EC01017=-23.5540,0.0000
EC01018=-21.4458,0.0000
EC01019=-19.3299,0.0000
EC01020=-17.2060,0.0000
EC01021=-15.2391,0.0000
EC01022=-13.7009,0.0000
EC01023=-12.7745,0.0000
EC01024=-12.0705,0.0000
EC01025=-11.3400,0.0000
EC01026=-10.3419,0.0000
EC01027=-8.6952,0.0000
EC01028=-6.0002,0.0000
EC01029=-3.0871,0.0000
EC01030=0.0000,0.0000
EC01031=0.0000,0.0000
EC01032=3.0565,0.0000
EC01033=5.9598,0.0000
EC01034=8.6610,0.0000
EC01035=10.2852,0.0000
EC01036=11.2483,0.0000
EC01037=11.9417,0.0000
EC01038=12.6030,0.0000
EC01039=13.4837,0.0000
EC01040=15.0155,0.0000
EC01041=17.0162,0.0000
EC01042=19.2050,0.0000
EC01043=21.4028,0.0000
EC01044=23.5971,0.0000
EC01045=25.7952,0.0000
EC01046=27.9837,0.0000
EC01047=29.9842,0.0000
EC01048=31.5162,0.0000
EC01049=32.3970,0.0000
EC01050=33.0583,0.0000
EC01051=33.7518,0.0000
EC01052=34.7152,0.0000
EC01053=36.3389,0.0000
EC01054=39.0399,0.0000
EC01055=41.9437,0.0000
EC01056=45.0000,0.0000
EC01057=48.0563,0.0000
EC01058=50.9601,0.0000
EC01059=53.6611,0.0000
EC01060=55.2848,0.0000
EC01061=56.2482,0.0000
EC01062=56.9417,0.0000
EC01063=57.6030,0.0000
EC01064=58.4838,0.0000
EC01065=60.0158,0.0000
EC01066=62.0163,0.0000
EC01067=64.2048,0.0000
EC01068=66.4029,0.0000
EC01069=68.5972,0.0000
EC01070=70.7950,0.0000
EC01071=72.9838,0.0000
EC01072=74.9845,0.0000
EC01073=76.5163,0.0000
EC01074=77.3970,0.0000
EC01075=78.0583,0.0000
EC01076=78.7517,0.0000
EC01077=79.7148,0.0000
EC01078=81.3390,0.0000
EC01079=84.0402,0.0000
EC01080=86.9435,0.0000
EC01081=90.0000,0.0000
EC01082=93.0565,0.0000
EC01083=95.9604,0.0000
EC01084=98.6610,0.0000
EC01085=100.2852,0.0000
EC01086=101.2483,0.0000
EC01087=101.9417,0.0000
EC01088=102.6030,0.0000
EC01089=103.4837,0.0000
EC01090=105.0155,0.0000
EC01091=107.0162,0.0000
EC01092=109.2050,0.0000
EC01093=111.4028,0.0000
EC01094=113.5971,0.0000
EC01095=115.7952,0.0000
EC01096=117.9837,0.0000
EC01097=119.9842,0.0000
EC01098=121.5162,0.0000
EC01099=122.3970,0.0000
EC01100=123.0583,0.0000
EC01101=123.7518,0.0000
EC01102=124.7152,0.0000
EC01103=126.3389,0.0000
EC01104=129.0399,0.0000
EC01105=131.9437,0.0000
EC01106=135.0000,0.0000
EC01107=138.0563,0.0000
EC01108=140.9601,0.0000
EC01109=143.6611,0.0000
EC01110=145.2848,0.0000
EC01111=146.2482,0.0000
EC01112=146.9417,0.0000
EC01113=147.6030,0.0000
EC01114=148.4838,0.0000
EC01115=150.0158,0.0000
EC01116=152.0163,0.0000
EC01117=154.2048,0.0000
EC01118=156.4029,0.0000
EC01119=158.5972,0.0000
EC01120=160.7950,0.0000
EC01121=162.9838,0.0000
EC01122=164.9845,0.0000
EC01123=166.5163,0.0000
EC01124=167.3970,0.0000
EC01125=168.0583,0.0000
EC01126=168.7517,0.0000
EC01127=169.7148,0.0000
EC01128=171.3390,0.0000
EC01129=174.0402,0.0000
EC01130=176.9435,0.0000
EC01131=180.0000,0.0000
EC01132=180.0000,0.0000
EC01133=-176.9435,0.0000
EC01134=-174.0396,0.0000
EC01135=-171.3390,0.0000
EC01136=-169.7148,0.0000
EC01137=-168.7517,0.0000
EC01138=-168.0583,0.0000
EC01139=-167.3970,0.0000
EC01140=-166.5163,0.0000
EC01141=-164.9845,0.0000
EC01142=-162.9838,0.0000
EC01143=-160.7950,0.0000
EC01144=-158.5972,0.0000
EC01145=-156.4029,0.0000
EC01146=-154.2048,0.0000
EC01147=-152.0163,0.0000
EC01148=-150.0158,0.0000
EC01149=-148.4838,0.0000
EC01150=-147.6030,0.0000
EC01151=-146.9417,0.0000
EC01152=-146.2482,0.0000
EC01153=-145.2848,0.0000
EC01154=-143.6611,0.0000
EC01155=-140.9601,0.0000
EC01156=-138.0563,0.0000
EC01157=-135.0000,0.0000
EC01158=-131.9437,0.0000
EC01159=-129.0399,0.0000
EC01160=-126.3389,0.0000
EC01161=-124.7152,0.0000
EC01162=-123.7518,0.0000
EC01163=-123.0583,0.0000
EC01164=-122.3970,0.0000
EC01165=-121.5162,0.0000
EC01166=-119.9842,0.0000
EC01167=-117.9837,0.0000
EC01168=-115.7952,0.0000
EC01169=-113.5971,0.0000
EC01170=-111.4028,0.0000
EC01171=-109.2050,0.0000
EC01172=-107.0162,0.0000
EC01173=-105.0155,0.0000
EC01174=-103.4837,0.0000
EC01175=-102.6030,0.0000
EC01176=-101.9417,0.0000
EC01177=-101.2483,0.0000
EC01178=-100.2852,0.0000
EC01179=-98.6610,0.0000
EC01180=-95.9598,0.0000
EC01181=-93.0565,0.0000
EC01182=-90.0000,0.0000
EC01183=-86.9435,0.0000
EC01184=-84.0396,0.0000
EC01185=-81.3390,0.0000
EC01186=-79.7148,0.0000
EC01187=-78.7517,0.0000
EC01188=-78.0583,0.0000
EC01189=-77.3970,0.0000
EC01190=-76.5163,0.0000
EC01191=-74.9845,0.0000
EC01192=-72.9838,0.0000
EC01193=-70.7950,0.0000
EC01194=-68.5972,0.0000
EC01195=-66.4029,0.0000
EC01196=-64.2048,0.0000
EC01197=-62.0163,0.0000
EC01198=-60.0158,0.0000
EC01199=-58.4838,0.0000
EC01200=-57.6030,0.0000
EC01201=-56.9417,0.0000
EC01202=-56.2482,0.0000
EC01203=-55.2848,0.0000
EC01204=-53.6611,0.0000
EC01205=-50.9601,0.0000
EC01206=-48.0563,0.0000
EC01207=-45.0000,0.0000
EC01208=-41.9437,0.0000
EC01209=-39.0399,0.0000
EC01210=-36.3389,0.0000
EC01211=-34.7152,0.0000
EC01212=-33.7518,0.0000
EC01213=-33.0583,0.0000
EC01214=-32.3970,0.0000
EC01215=-31.5162,0.0000
EC01216=-29.9842,0.0000
EC01217=-27.9837,0.0000
EC01218=-25.7952,0.0000
EC01219=-23.5971,0.0000
EC01220=-21.4028,0.0000
EC01221=-19.2050,0.0000
EC01222=-17.0162,0.0000
EC01223=-15.0155,0.0000
EC01224=-13.4837,0.0000
EC01225=-12.6030,0.0000
EC01226=-11.9417,0.0000
EC01227=-11.2483,0.0000
EC01228=-10.2852,0.0000
EC01229=-8.6610,0.0000
EC01230=-5.9604,0.0000
EC01231=-3.0565,0.0000
EC01232=0.0000,0.0000
EC01233=0.0000,0.0000
EC01234=3.0242,0.0000
EC01235=5.9175,0.0000
EC01236=8.6252,0.0000
EC01237=10.2250,0.0000
EC01238=11.1519,0.0000
EC01239=11.8065,0.0000
EC01240=12.4248,0.0000
EC01241=13.2580,0.0000
EC01242=14.7847,0.0000
EC01243=16.8204,0.0000
EC01244=19.0758,0.0000
EC01245=21.3580,0.0000
EC01246=23.6417,0.0000
EC01247=25.9241,0.0000
EC01248=28.1796,0.0000
EC01249=30.2155,0.0000
EC01250=31.7418,0.0000
EC01251=32.5751,0.0000
EC01252=33.1936,0.0000
EC01253=33.8475,0.0000
EC01254=34.7753,0.0000
EC01255=36.3747,0.0000
EC01256=39.0826,0.0000
EC01257=41.9754,0.0000
EC01258=45.0000,0.0000
EC01259=48.0237,0.0000
EC01260=50.9174,0.0000
EC01261=53.6253,0.0000
EC01262=55.2247,0.0000
EC01263=56.1525,0.0000
EC01264=56.8064,0.0000
EC01265=57.4249,0.0000
EC01266=58.2582,0.0000
EC01267=59.7845,0.0000
EC01268=61.8204,0.0000
EC01269=64.0759,0.0000
EC01270=66.3583,0.0000
EC01271=68.6420,0.0000
EC01272=70.9242,0.0000
EC01273=73.1796,0.0000
EC01274=75.2153,0.0000
EC01275=76.7420,0.0000
EC01276=77.5752,0.0000
EC01277=78.1935,0.0000
EC01278=78.8481,0.0000
EC01279=79.7750,0.0000
EC01280=81.3748,0.0000
EC01281=84.0825,0.0000
EC01282=86.9758,0.0000
EC01283=90.0000,0.0000
EC01284=93.0242,0.0000
EC01285=95.9175,0.0000
EC01286=98.6252,0.0000
EC01287=100.2250,0.0000
EC01288=101.1519,0.0000
EC01289=101.8065,0.0000
EC01290=102.4248,0.0000
EC01291=103.2580,0.0000
EC01292=104.7847,0.0000
EC01293=106.8204,0.0000
EC01294=109.0758,0.0000
EC01295=111.3580,0.0000
EC01296=113.6417,0.0000
EC01297=115.9241,0.0000
EC01298=118.1796,0.0000
EC01299=120.2155,0.0000
EC01300=121.7418,0.0000
EC01301=122.5751,0.0000
EC01302=123.1936,0.0000
EC01303=123.8475,0.0000
EC01304=124.7753,0.0000
EC01305=126.3747,0.0000
EC01306=129.0826,0.0000
EC01307=131.9754,0.0000
EC01308=135.0000,0.0000
EC01309=138.0237,0.0000
EC01310=140.9174,0.0000
EC01311=143.6253,0.0000
EC01312=145.2247,0.0000
EC01313=146.1525,0.0000
EC01314=146.8064,0.0000
EC01315=147.4249,0.0000
EC01316=148.2582,0.0000
EC01317=149.7845,0.0000
EC01318=151.8204,0.0000
EC01319=154.0759,0.0000
EC01320=156.3583,0.0000
EC01321=158.6420,0.0000
EC01322=160.9242,0.0000
EC01323=163.1796,0.0000
EC01324=165.2153,0.0000
EC01325=166.7420,0.0000
EC01326=167.5752,0.0000
EC01327=168.1935,0.0000
EC01328=168.8481,0.0000
EC01329=169.7750,0.0000
EC01330=171.3748,0.0000
EC01331=174.0825,0.0000
EC01332=176.9758,0.0000
EC01333=180.0000,0.0000
EC01334=180.0000,0.0000
EC01335=-176.9758,0.0000
EC01336=-174.0825,0.0000
EC01337=-171.3748,0.0000
EC01338=-169.7750,0.0000
EC01339=-168.8481,0.0000
EC01340=-168.1935,0.0000
EC01341=-167.5752,0.0000
EC01342=-166.7420,0.0000
EC01343=-165.2153,0.0000
EC01344=-163.1796,0.0000
EC01345=-160.9242,0.0000
EC01346=-158.6420,0.0000
EC01347=-156.3583,0.0000
EC01348=-154.0759,0.0000
EC01349=-151.8204,0.0000
EC01350=-149.7845,0.0000
EC01351=-148.2582,0.0000
EC01352=-147.4249,0.0000
EC01353=-146.8064,0.0000
EC01354=-146.1525,0.0000
EC01355=-145.2247,0.0000
EC01356=-143.6253,0.0000
EC01357=-140.9174,0.0000
EC01358=-138.0246,0.0000
EC01359=-135.0000,0.0000
EC01360=-131.9763,0.0000
EC01361=-129.0826,0.0000
EC01362=-126.3747,0.0000
EC01363=-124.7753,0.0000
EC01364=-123.8475,0.0000
EC01365=-123.1936,0.0000
EC01366=-122.5751,0.0000
EC01367=-121.7418,0.0000
EC01368=-120.2155,0.0000
EC01369=-118.1796,0.0000
EC01370=-115.9241,0.0000
EC01371=-113.6417,0.0000
EC01372=-111.3580,0.0000
EC01373=-109.0758,0.0000
EC01374=-106.8204,0.0000
EC01375=-104.7847,0.0000
EC01376=-103.2580,0.0000
EC01377=-102.4248,0.0000
EC01378=-101.8065,0.0000
EC01379=-101.1519,0.0000
EC01380=-100.2250,0.0000
EC01381=-98.6252,0.0000
EC01382=-95.9175,0.0000
EC01383=-93.0242,0.0000
EC01384=-90.0000,0.0000
EC01385=-86.9758,0.0000
EC01386=-84.0825,0.0000
EC01387=-81.3748,0.0000
EC01388=-79.7750,0.0000
EC01389=-78.8481,0.0000
EC01390=-78.1935,0.0000
EC01391=-77.5752,0.0000
EC01392=-76.7420,0.0000
EC01393=-75.2153,0.0000
EC01394=-73.1796,0.0000
EC01395=-70.9242,0.0000
EC01396=-68.6420,0.0000
EC01397=-66.3583,0.0000
EC01398=-64.0759,0.0000
EC01399=-61.8204,0.0000
EC01400=-59.7845,0.0000
EC01401=-58.2582,0.0000
EC01402=-57.4249,0.0000
EC01403=-56.8064,0.0000
EC01404=-56.1525,0.0000
EC01405=-55.2247,0.0000
EC01406=-53.6253,0.0000
EC01407=-50.9174,0.0000
EC01408=-48.0246,0.0000
EC01409=-45.0000,0.0000
EC01410=-41.9763,0.0000
EC01411=-39.0826,0.0000
EC01412=-36.3747,0.0000
EC01413=-34.7753,0.0000
EC01414=-33.8475,0.0000
EC01415=-33.1936,0.0000
EC01416=-32.5751,0.0000
EC01417=-31.7418,0.0000
EC01418=-30.2155,0.0000
EC01419=-28.1796,0.0000
EC01420=-25.9241,0.0000
EC01421=-23.6417,0.0000
EC01422=-21.3580,0.0000
EC01423=-19.0758,0.0000
EC01424=-16.8204,0.0000
EC01425=-14.7847,0.0000
EC01426=-13.2580,0.0000
EC01427=-12.4248,0.0000
EC01428=-11.8065,0.0000
EC01429=-11.1519,0.0000
EC01430=-10.2250,0.0000
EC01431=-8.6252,0.0000
EC01432=-5.9175,0.0000
EC01433=-3.0242,0.0000
EC01434=0.0000,0.0000
EC01435=0.0000,0.0000
EC01436=2.9903,0.0000
EC01437=5.8729,0.0000
EC01438=8.5881,0.0000
EC01439=10.1621,0.0000
EC01440=11.0515,0.0000
EC01441=11.6656,0.0000
EC01442=12.2395,0.0000
EC01443=13.0258,0.0000
EC01444=14.5467,0.0000
EC01445=16.6187,0.0000
EC01446=18.9437,0.0000
EC01447=21.3119,0.0000
EC01448=23.6874,0.0000
EC01449=26.0569,0.0000
EC01450=28.3812,0.0000
EC01451=30.4534,0.0000
EC01452=31.9748,0.0000
EC01453=32.7607,0.0000
EC01454=33.3343,0.0000
EC01455=33.9482,0.0000
EC01456=34.8381,0.0000
EC01457=36.4120,0.0000
EC01458=39.1268,0.0000
EC01459=42.0095,0.0000
EC01460=45.0000,0.0000
EC01461=47.9905,0.0000
EC01462=50.8732,0.0000
EC01463=53.5880,0.0000
EC01464=55.1619,0.0000
EC01465=56.0518,0.0000
EC01466=56.6657,0.0000
EC01467=57.2393,0.0000
EC01468=58.0252,0.0000
EC01469=59.5466,0.0000
EC01470=61.6188,0.0000
EC01471=63.9431,0.0000
EC01472=66.3126,0.0000
EC01473=68.6881,0.0000
EC01474=71.0563,0.0000
EC01475=73.3813,0.0000
EC01476=75.4533,0.0000
EC01477=76.9742,0.0000
EC01478=77.7605,0.0000
EC01479=78.3344,0.0000
EC01480=78.9485,0.0000
EC01481=79.8379,0.0000
EC01482=81.4119,0.0000
EC01483=84.1271,0.0000
EC01484=87.0097,0.0000
EC01485=90.0000,0.0000
EC01486=92.9903,0.0000
EC01487=95.8729,0.0000
EC01488=98.5881,0.0000
EC01489=100.1621,0.0000
EC01490=101.0515,0.0000
EC01491=101.6656,0.0000
EC01492=102.2395,0.0000
EC01493=103.0258,0.0000
EC01494=104.5467,0.0000
EC01495=106.6187,0.0000
EC01496=108.9437,0.0000
EC01497=111.3119,0.0000
EC01498=113.6874,0.0000
EC01499=116.0569,0.0000
EC01500=118.3812,0.0000
EC01501=120.4534,0.0000
EC01502=121.9748,0.0000
EC01503=122.7607,0.0000
EC01504=123.3343,0.0000
EC01505=123.9482,0.0000
EC01506=124.8381,0.0000
EC01507=126.4120,0.0000
EC01508=129.1268,0.0000
EC01509=132.0095,0.0000
EC01510=135.0000,0.0000
EC01511=137.9905,0.0000
EC01512=140.8732,0.0000
EC01513=143.5880,0.0000
EC01514=145.1619,0.0000
EC01515=146.0518,0.0000
EC01516=146.6657,0.0000
EC01517=147.2393,0.0000
EC01518=148.0252,0.0000
EC01519=149.5466,0.0000
EC01520=151.6188,0.0000
EC01521=153.9431,0.0000
EC01522=156.3126,0.0000
EC01523=158.6881,0.0000
EC01524=161.0563,0.0000
EC01525=163.3813,0.0000
EC01526=165.4533,0.0000
EC01527=166.9742,0.0000
EC01528=167.7605,0.0000
EC01529=168.3344,0.0000
EC01530=168.9485,0.0000
EC01531=169.8379,0.0000
EC01532=171.4119,0.0000
EC01533=174.1271,0.0000
EC01534=177.0097,0.0000
EC01535=180.0000,0.0000
EC01536=180.0000,0.0000
EC01537=-177.0097,0.0000
EC01538=-174.1271,0.0000
EC01539=-171.4119,0.0000
EC01540=-169.8379,0.0000
EC01541=-168.9485,0.0000
EC01542=-168.3344,0.0000
EC01543=-167.7605,0.0000
EC01544=-166.9742,0.0000
EC01545=-165.4533,0.0000
EC01546=-163.3813,0.0000
EC01547=-161.0563,0.0000
EC01548=-158.6881,0.0000
EC01549=-156.3126,0.0000
EC01550=-153.9431,0.0000
EC01551=-151.6188,0.0000
EC01552=-149.5466,0.0000
EC01553=-148.0252,0.0000
EC01554=-147.2393,0.0000
EC01555=-146.6657,0.0000
EC01556=-146.0518,0.0000
EC01557=-145.1619,0.0000
EC01558=-143.5880,0.0000
EC01559=-140.8732,0.0000
EC01560=-137.9905,0.0000
EC01561=-135.0000,0.0000
EC01562=-132.0095,0.0000
EC01563=-129.1268,0.0000
EC01564=-126.4120,0.0000
EC01565=-124.8381,0.0000
EC01566=-123.9482,0.0000
EC01567=-123.3343,0.0000
EC01568=-122.7607,0.0000
EC01569=-121.9748,0.0000
EC01570=-120.4534,0.0000
EC01571=-118.3812,0.0000
EC01572=-116.0569,0.0000
EC01573=-113.6874,0.0000
EC01574=-111.3119,0.0000
EC01575=-108.9437,0.0000
EC01576=-106.6187,0.0000
EC01577=-104.5467,0.0000
EC01578=-103.0258,0.0000
EC01579=-102.2395,0.0000
EC01580=-101.6656,0.0000
EC01581=-101.0515,0.0000
EC01582=-100.1621,0.0000
EC01583=-98.5881,0.0000
EC01584=-95.8729,0.0000
EC01585=-92.9903,0.0000
EC01586=-90.0000,0.0000
EC01587=-87.0097,0.0000
EC01588=-84.1271,0.0000
EC01589=-81.4119,0.0000
EC01590=-79.8379,0.0000
EC01591=-78.9485,0.0000
EC01592=-78.3344,0.0000
EC01593=-77.7605,0.0000
EC01594=-76.9742,0.0000
EC01595=-75.4533,0.0000
EC01596=-73.3813,0.0000
EC01597=-71.0563,0.0000
EC01598=-68.6881,0.0000
EC01599=-66.3126,0.0000
EC01600=-63.9431,0.0000
EC01601=-61.6188,0.0000
EC01602=-59.5466,0.0000
EC01603=-58.0252,0.0000
EC01604=-57.2393,0.0000
EC01605=-56.6657,0.0000
EC01606=-56.0518,0.0000
EC01607=-55.1619,0.0000
EC01608=-53.5880,0.0000
EC01609=-50.8732,0.0000
EC01610=-47.9905,0.0000
EC01611=-45.0000,0.0000
EC01612=-42.0095,0.0000
EC01613=-39.1268,0.0000
EC01614=-36.4120,0.0000
EC01615=-34.8381,0.0000
EC01616=-33.9482,0.0000
EC01617=-33.3343,0.0000
EC01618=-32.7607,0.0000
EC01619=-31.9748,0.0000
EC01620=-30.4534,0.0000
EC01621=-28.3812,0.0000
EC01622=-26.0569,0.0000
EC01623=-23.6874,0.0000
EC01624=-21.3119,0.0000
EC01625=-18.9437,0.0000
EC01626=-16.6187,0.0000
EC01627=-14.5467,0.0000
EC01628=-13.0258,0.0000
EC01629=-12.2395,0.0000
EC01630=-11.6656,0.0000
EC01631=-11.0515,0.0000
EC01632=-10.1621,0.0000
EC01633=-8.5881,0.0000
EC01634=-5.8729,0.0000
EC01635=-2.9903,0.0000
EC01636=0.0000,0.0000
EC01637=0.0000,0.0000
EC01638=2.9548,0.0000
EC01639=5.8263,0.0000
EC01640=8.5486,0.0000
EC01641=10.0964,0.0000
EC01642=10.9471,0.0000
EC01643=11.5198,0.0000
EC01644=12.0484,0.0000
EC01645=12.7860,0.0000
EC01646=14.3034,0.0000
EC01647=16.4132,0.0000
EC01648=18.8079,0.0000
EC01649=21.2653,0.0000
EC01650=23.7346,0.0000
EC01651=26.1917,0.0000
EC01652=28.5867,0.0000
EC01653=30.6966,0.0000
EC01654=32.2136,0.0000
EC01655=32.9519,0.0000
EC01656=33.4806,0.0000
EC01657=34.0527,0.0000
EC01658=34.9034,0.0000
EC01659=36.4513,0.0000
EC01660=39.1737,0.0000
EC01661=42.0450,0.0000
EC01662=45.0000,0.0000
EC01663=47.9550,0.0000
EC01664=50.8263,0.0000
EC01665=53.5487,0.0000
EC01666=55.0966,0.0000
EC01667=55.9473,0.0000
EC01668=56.5194,0.0000
EC01669=57.0481,0.0000
EC01670=57.7864,0.0000
EC01671=59.3034,0.0000
EC01672=61.4133,0.0000
EC01673=63.8083,0.0000
EC01674=66.2654,0.0000
EC01675=68.7347,0.0000
EC01676=71.1921,0.0000
EC01677=73.5868,0.0000
EC01678=75.6966,0.0000
EC01679=77.2140,0.0000
EC01680=77.9516,0.0000
EC01681=78.4802,0.0000
EC01682=79.0529,0.0000
EC01683=79.9036,0.0000
EC01684=81.4514,0.0000
EC01685=84.1737,0.0000
EC01686=87.0452,0.0000
EC01687=90.0000,0.0000
EC01688=92.9548,0.0000
EC01689=95.8263,0.0000
EC01690=98.5486,0.0000
EC01691=100.0964,0.0000
EC01692=100.9471,0.0000
EC01693=101.5198,0.0000
EC01694=102.0484,0.0000
EC01695=102.7860,0.0000
EC01696=104.3034,0.0000
EC01697=106.4132,0.0000
EC01698=108.8079,0.0000
EC01699=111.2653,0.0000
EC01700=113.7346,0.0000
EC01701=116.1917,0.0000
EC01702=118.5867,0.0000
EC01703=120.6966,0.0000
EC01704=122.2136,0.0000
EC01705=122.9519,0.0000
EC01706=123.4806,0.0000
EC01707=124.0527,0.0000
EC01708=124.9034,0.0000
EC01709=126.4513,0.0000
EC01710=129.1737,0.0000
EC01711=132.0450,0.0000
EC01712=135.0000,0.0000
EC01713=137.9550,0.0000
EC01714=140.8263,0.0000
EC01715=143.5487,0.0000
EC01716=145.0966,0.0000
EC01717=145.9473,0.0000
EC01718=146.5194,0.0000
EC01719=147.0481,0.0000
EC01720=147.7864,0.0000
EC01721=149.3034,0.0000
EC01722=151.4133,0.0000
EC01723=153.8083,0.0000
EC01724=156.2654,0.0000
EC01725=158.7347,0.0000
EC01726=161.1921,0.0000
EC01727=163.5868,0.0000
EC01728=165.6966,0.0000
EC01729=167.2140,0.0000
EC01730=167.9516,0.0000
EC01731=168.4802,0.0000
EC01732=169.0529,0.0000
EC01733=169.9036,0.0000
EC01734=171.4514,0.0000
EC01735=174.1737,0.0000
EC01736=177.0452,0.0000
EC01737=180.0000,0.0000
EC01738=180.0000,0.0000
EC01739=-177.0452,0.0000
EC01740=-174.1737,0.0000
EC01741=-171.4514,0.0000
EC01742=-169.9036,0.0000
EC01743=-169.0529,0.0000
EC01744=-168.4802,0.0000
EC01745=-167.9516,0.0000
EC01746=-167.2140,0.0000
EC01747=-165.6966,0.0000
EC01748=-163.5868,0.0000
EC01749=-161.1921,0.0000
EC01750=-158.7347,0.0000
EC01751=-156.2654,0.0000
EC01752=-153.8083,0.0000
EC01753=-151.4133,0.0000
EC01754=-149.3034,0.0000
EC01755=-147.7864,0.0000
EC01756=-147.0481,0.0000
EC01757=-146.5194,0.0000
EC01758=-145.9473,0.0000
EC01759=-145.0966,0.0000
EC01760=-143.5487,0.0000
EC01761=-140.8263,0.0000
EC01762=-137.9550,0.0000
EC01763=-135.0000,0.0000
EC01764=-132.0450,0.0000
EC01765=-129.1737,0.0000
EC01766=-126.4513,0.0000
EC01767=-124.9034,0.0000
EC01768=-124.0527,0.0000
EC01769=-123.4806,0.0000
EC01770=-122.9519,0.0000
EC01771=-122.2136,0.0000
EC01772=-120.6966,0.0000
EC01773=-118.5867,0.0000
EC01774=-116.1917,0.0000
EC01775=-113.7346,0.0000
EC01776=-111.2653,0.0000
EC01777=-108.8079,0.0000
EC01778=-106.4132,0.0000
EC01779=-104.3034,0.0000
EC01780=-102.7860,0.0000
EC01781=-102.0484,0.0000
EC01782=-101.5198,0.0000
EC01783=-100.9471,0.0000
EC01784=-100.0964,0.0000
EC01785=-98.5486,0.0000
EC01786=-95.8263,0.0000
EC01787=-92.9548,0.0000
EC01788=-90.0000,0.0000
EC01789=-87.0452,0.0000
EC01790=-84.1737,0.0000
EC01791=-81.4514,0.0000
EC01792=-79.9036,0.0000
EC01793=-79.0529,0.0000
EC01794=-78.4802,0.0000
EC01795=-77.9516,0.0000
EC01796=-77.2140,0.0000
EC01797=-75.6966,0.0000
EC01798=-73.5868,0.0000
EC01799=-71.1921,0.0000
EC01800=-68.7347,0.0000
EC01801=-66.2654,0.0000
EC01802=-63.8083,0.0000
EC01803=-61.4133,0.0000
EC01804=-59.3034,0.0000
EC01805=-57.7864,0.0000
EC01806=-57.0481,0.0000
EC01807=-56.5194,0.0000
EC01808=-55.9473,0.0000
EC01809=-55.0966,0.0000
EC01810=-53.5487,0.0000
EC01811=-50.8263,0.0000
EC01812=-47.9550,0.0000
EC01813=-45.0000,0.0000
EC01814=-42.0450,0.0000
EC01815=-39.1737,0.0000
EC01816=-36.4513,0.0000
EC01817=-34.9034,0.0000
EC01818=-34.0527,0.0000
EC01819=-33.4806,0.0000
EC01820=-32.9519,0.0000
EC01821=-32.2136,0.0000
EC01822=-30.6966,0.0000
EC01823=-28.5867,0.0000
EC01824=-26.1917,0.0000
EC01825=-23.7346,0.0000
EC01826=-21.2653,0.0000
EC01827=-18.8079,0.0000
EC01828=-16.4132,0.0000
EC01829=-14.3034,0.0000
EC01830=-12.7860,0.0000
EC01831=-12.0484,0.0000
EC01832=-11.5198,0.0000
EC01833=-10.9471,0.0000
EC01834=-10.0964,0.0000
EC01835=-8.5486,0.0000
EC01836=-5.8263,0.0000
EC01837=-2.9548,0.0000
EC01838=0.0000,0.0000
EC01839=0.0000,0.0000
EC01840=2.9180,0.0000
EC01841=5.7775,0.0000
EC01842=8.5076,0.0000
EC01843=10.0280,0.0000
EC01844=10.8382,0.0000
EC01845=11.3683,0.0000
EC01846=11.8512,0.0000
EC01847=12.5410,0.0000
EC01848=14.0550,0.0000
EC01849=16.2037,0.0000
EC01850=18.6701,0.0000
EC01851=21.2180,0.0000
EC01852=23.7821,0.0000
EC01853=26.3297,0.0000
EC01854=28.7961,0.0000
EC01855=30.9450,0.0000
EC01856=32.4587,0.0000
EC01857=33.1487,0.0000
EC01858=33.6320,0.0000
EC01859=34.1614,0.0000
EC01860=34.9722,0.0000
EC01861=36.4919,0.0000
EC01862=39.2230,0.0000
EC01863=42.0820,0.0000
EC01864=45.0000,0.0000
EC01865=47.9180,0.0000
EC01866=50.7770,0.0000
EC01867=53.5081,0.0000
EC01868=55.0278,0.0000
EC01869=55.8386,0.0000
EC01870=56.3680,0.0000
EC01871=56.8513,0.0000
EC01872=57.5413,0.0000
EC01873=59.0550,0.0000
EC01874=61.2039,0.0000
EC01875=63.6703,0.0000
EC01876=66.2179,0.0000
EC01877=68.7820,0.0000
EC01878=71.3299,0.0000
EC01879=73.7963,0.0000
EC01880=75.9450,0.0000
EC01881=77.4590,0.0000
EC01882=78.1488,0.0000
EC01883=78.6317,0.0000
EC01884=79.1618,0.0000
EC01885=79.9720,0.0000
EC01886=81.4924,0.0000
EC01887=84.2225,0.0000
EC01888=87.0820,0.0000
EC01889=90.0000,0.0000
EC01890=92.9180,0.0000
EC01891=95.7775,0.0000
EC01892=98.5076,0.0000
EC01893=100.0280,0.0000
EC01894=100.8382,0.0000
EC01895=101.3683,0.0000
EC01896=101.8512,0.0000
EC01897=102.5410,0.0000
EC01898=104.0550,0.0000
EC01899=106.2037,0.0000
EC01900=108.6701,0.0000
EC01901=111.2180,0.0000
EC01902=113.7821,0.0000
EC01903=116.3297,0.0000
EC01904=118.7961,0.0000
EC01905=120.9450,0.0000
EC01906=122.4587,0.0000
EC01907=123.1487,0.0000
EC01908=123.6320,0.0000
EC01909=124.1614,0.0000
EC01910=124.9722,0.0000
EC01911=126.4919,0.0000
EC01912=129.2230,0.0000
EC01913=132.0820,0.0000
EC01914=135.0000,0.0000
EC01915=137.9180,0.0000
EC01916=140.7770,0.0000
EC01917=143.5081,0.0000
EC01918=145.0278,0.0000
EC01919=145.8386,0.0000
EC01920=146.3680,0.0000
EC01921=146.8513,0.0000
EC01922=147.5413,0.0000
EC01923=149.0550,0.0000
EC01924=151.2039,0.0000
EC01925=153.6703,0.0000
EC01926=156.2179,0.0000
EC01927=158.7820,0.0000
EC01928=161.3299,0.0000
EC01929=163.7963,0.0000
EC01930=165.9450,0.0000
EC01931=167.4590,0.0000
EC01932=168.1488,0.0000
EC01933=168.6317,0.0000
EC01934=169.1618,0.0000
EC01935=169.9720,0.0000
EC01936=171.4924,0.0000
EC01937=174.2225,0.0000
EC01938=177.0820,0.0000
EC01939=180.0000,0.0000
EC01940=180.0000,0.0000
EC01941=-177.0820,0.0000
EC01942=-174.2225,0.0000
EC01943=-171.4924,0.0000
EC01944=-169.9720,0.0000
EC01945=-169.1618,0.0000
EC01946=-168.6317,0.0000
EC01947=-168.1488,0.0000
EC01948=-167.4590,0.0000
EC01949=-165.9450,0.0000
EC01950=-163.7963,0.0000
EC01951=-161.3299,0.0000
EC01952=-158.7820,0.0000
EC01953=-156.2179,0.0000
EC01954=-153.6703,0.0000
EC01955=-151.2039,0.0000
EC01956=-149.0550,0.0000
EC01957=-147.5413,0.0000
EC01958=-146.8513,0.0000
EC01959=-146.3680,0.0000
EC01960=-145.8386,0.0000
EC01961=-145.0278,0.0000
EC01962=-143.5081,0.0000
EC01963=-140.7770,0.0000
EC01964=-137.9180,0.0000
EC01965=-135.0000,0.0000
EC01966=-132.0820,0.0000
EC01967=-129.2230,0.0000
EC01968=-126.4919,0.0000
EC01969=-124.9722,0.0000
EC01970=-124.1614,0.0000
EC01971=-123.6320,0.0000
EC01972=-123.1487,0.0000
EC01973=-122.4587,0.0000
EC01974=-120.9450,0.0000
EC01975=-118.7961,0.0000
EC01976=-116.3297,0.0000
EC01977=-113.7821,0.0000
EC01978=-111.2180,0.0000
EC01979=-108.6701,0.0000
EC01980=-106.2037,0.0000
EC01981=-104.0550,0.0000
EC01982=-102.5410,0.0000
EC01983=-101.8512,0.0000
EC01984=-101.3683,0.0000
EC01985=-100.8382,0.0000
EC01986=-100.0280,0.0000
EC01987=-98.5076,0.0000
EC01988=-95.7775,0.0000
EC01989=-92.9180,0.0000
EC01990=-90.0000,0.0000
EC01991=-87.0820,0.0000
EC01992=-84.2225,0.0000
EC01993=-81.4924,0.0000
EC01994=-79.9720,0.0000
EC01995=-79.1618,0.0000
EC01996=-78.6317,0.0000
EC01997=-78.1488,0.0000
EC01998=-77.4590,0.0000
EC01999=-75.9450,0.0000
//INST
///DATE 2021/02/10 13:51
///COMM
///ATTR SC,RW,RJ
////FRAME USER 2
///GROUP1 RB1
///GROUP2 ST1
NOP
SMOVL C00000 +MOVJ EC00000
SMOVL C00001 +MOVJ EC00001
SMOVL C00002 +MOVJ EC00002
SMOVL C00003 +MOVJ EC00003
SMOVL C00004 +MOVJ EC00004
SMOVL C00005 +MOVJ EC00005
SMOVL C00006 +MOVJ EC00006
SMOVL C00007 +MOVJ EC00007
SMOVL C00008 +MOVJ EC00008
SMOVL C00009 +MOVJ EC00009
SMOVL C00010 +MOVJ EC00010
SMOVL C00011 +MOVJ EC00011
SMOVL C00012 +MOVJ EC00012
SMOVL C00013 +MOVJ EC00013
SMOVL C00014 +MOVJ EC00014
SMOVL C00015 +MOVJ EC00015
SMOVL C00016 +MOVJ EC00016
SMOVL C00017 +MOVJ EC00017
SMOVL C00018 +MOVJ EC00018
SMOVL C00019 +MOVJ EC00019
SMOVL C00020 +MOVJ EC00020
SMOVL C00021 +MOVJ EC00021
SMOVL C00022 +MOVJ EC00022
SMOVL C00023 +MOVJ EC00023
SMOVL C00024 +MOVJ EC00024
SMOVL C00025 +MOVJ EC00025
SMOVL C00026 +MOVJ EC00026
SMOVL C00027 +MOVJ EC00027
SMOVL C00028 +MOVJ EC00028
SMOVL C00029 +MOVJ EC00029
SMOVL C00030 +MOVJ EC00030
SMOVL C00031 +MOVJ EC00031
SMOVL C00032 +MOVJ EC00032
SMOVL C00033 +MOVJ EC00033
SMOVL C00034 +MOVJ EC00034
SMOVL C00035 +MOVJ EC00035
SMOVL C00036 +MOVJ EC00036
SMOVL C00037 +MOVJ EC00037
SMOVL C00038 +MOVJ EC00038
SMOVL C00039 +MOVJ EC00039
SMOVL C00040 +MOVJ EC00040
SMOVL C00041 +MOVJ EC00041
SMOVL C00042 +MOVJ EC00042
SMOVL C00043 +MOVJ EC00043
SMOVL C00044 +MOVJ EC00044
SMOVL C00045 +MOVJ EC00045
SMOVL C00046 +MOVJ EC00046
SMOVL C00047 +MOVJ EC00047
SMOVL C00048 +MOVJ EC00048
SMOVL C00049 +MOVJ EC00049
SMOVL C00050 +MOVJ EC00050
SMOVL C00051 +MOVJ EC00051
SMOVL C00052 +MOVJ EC00052
SMOVL C00053 +MOVJ EC00053
SMOVL C00054 +MOVJ EC00054
SMOVL C00055 +MOVJ EC00055
SMOVL C00056 +MOVJ EC00056
SMOVL C00057 +MOVJ EC00057
SMOVL C00058 +MOVJ EC00058
SMOVL C00059 +MOVJ EC00059
SMOVL C00060 +MOVJ EC00060
SMOVL C00061 +MOVJ EC00061
SMOVL C00062 +MOVJ EC00062
SMOVL C00063 +MOVJ EC00063
SMOVL C00064 +MOVJ EC00064
SMOVL C00065 +MOVJ EC00065
SMOVL C00066 +MOVJ EC00066
SMOVL C00067 +MOVJ EC00067
SMOVL C00068 +MOVJ EC00068
SMOVL C00069 +MOVJ EC00069
SMOVL C00070 +MOVJ EC00070
SMOVL C00071 +MOVJ EC00071
SMOVL C00072 +MOVJ EC00072
SMOVL C00073 +MOVJ EC00073
SMOVL C00074 +MOVJ EC00074
SMOVL C00075 +MOVJ EC00075
SMOVL C00076 +MOVJ EC00076
SMOVL C00077 +MOVJ EC00077
SMOVL C00078 +MOVJ EC00078
SMOVL C00079 +MOVJ EC00079
SMOVL C00080 +MOVJ EC00080
SMOVL C00081 +MOVJ EC00081
SMOVL C00082 +MOVJ EC00082
SMOVL C00083 +MOVJ EC00083
SMOVL C00084 +MOVJ EC00084
SMOVL C00085 +MOVJ EC00085
SMOVL C00086 +MOVJ EC00086
SMOVL C00087 +MOVJ EC00087
SMOVL C00088 +MOVJ EC00088
SMOVL C00089 +MOVJ EC00089
SMOVL C00090 +MOVJ EC00090
SMOVL C00091 +MOVJ EC00091
SMOVL C00092 +MOVJ EC00092
SMOVL C00093 +MOVJ EC00093
SMOVL C00094 +MOVJ EC00094
SMOVL C00095 +MOVJ EC00095
SMOVL C00096 +MOVJ EC00096
SMOVL C00097 +MOVJ EC00097
SMOVL C00098 +MOVJ EC00098
SMOVL C00099 +MOVJ EC00099
SMOVL C00100 +MOVJ EC00100
SMOVL C00101 +MOVJ EC00101
SMOVL C00102 +MOVJ EC00102
SMOVL C00103 +MOVJ EC00103
SMOVL C00104 +MOVJ EC00104
SMOVL C00105 +MOVJ EC00105
SMOVL C00106 +MOVJ EC00106
SMOVL C00107 +MOVJ EC00107
SMOVL C00108 +MOVJ EC00108
SMOVL C00109 +MOVJ EC00109
SMOVL C00110 +MOVJ EC00110
SMOVL C00111 +MOVJ EC00111
SMOVL C00112 +MOVJ EC00112
SMOVL C00113 +MOVJ EC00113
SMOVL C00114 +MOVJ EC00114
SMOVL C00115 +MOVJ EC00115
SMOVL C00116 +MOVJ EC00116
SMOVL C00117 +MOVJ EC00117
SMOVL C00118 +MOVJ EC00118
SMOVL C00119 +MOVJ EC00119
SMOVL C00120 +MOVJ EC00120
SMOVL C00121 +MOVJ EC00121
SMOVL C00122 +MOVJ EC00122
SMOVL C00123 +MOVJ EC00123
SMOVL C00124 +MOVJ EC00124
SMOVL C00125 +MOVJ EC00125
SMOVL C00126 +MOVJ EC00126
SMOVL C00127 +MOVJ EC00127
SMOVL C00128 +MOVJ EC00128
SMOVL C00129 +MOVJ EC00129
SMOVL C00130 +MOVJ EC00130
SMOVL C00131 +MOVJ EC00131
SMOVL C00132 +MOVJ EC00132
SMOVL C00133 +MOVJ EC00133
SMOVL C00134 +MOVJ EC00134
SMOVL C00135 +MOVJ EC00135
SMOVL C00136 +MOVJ EC00136
SMOVL C00137 +MOVJ EC00137
SMOVL C00138 +MOVJ EC00138
SMOVL C00139 +MOVJ EC00139
SMOVL C00140 +MOVJ EC00140
SMOVL C00141 +MOVJ EC00141
SMOVL C00142 +MOVJ EC00142
SMOVL C00143 +MOVJ EC00143
SMOVL C00144 +MOVJ EC00144
SMOVL C00145 +MOVJ EC00145
SMOVL C00146 +MOVJ EC00146
SMOVL C00147 +MOVJ EC00147
SMOVL C00148 +MOVJ EC00148
SMOVL C00149 +MOVJ EC00149
SMOVL C00150 +MOVJ EC00150
SMOVL C00151 +MOVJ EC00151
SMOVL C00152 +MOVJ EC00152
SMOVL C00153 +MOVJ EC00153
SMOVL C00154 +MOVJ EC00154
SMOVL C00155 +MOVJ EC00155
SMOVL C00156 +MOVJ EC00156
SMOVL C00157 +MOVJ EC00157
SMOVL C00158 +MOVJ EC00158
SMOVL C00159 +MOVJ EC00159
SMOVL C00160 +MOVJ EC00160
SMOVL C00161 +MOVJ EC00161
SMOVL C00162 +MOVJ EC00162
SMOVL C00163 +MOVJ EC00163
SMOVL C00164 +MOVJ EC00164
SMOVL C00165 +MOVJ EC00165
SMOVL C00166 +MOVJ EC00166
SMOVL C00167 +MOVJ EC00167
SMOVL C00168 +MOVJ EC00168
SMOVL C00169 +MOVJ EC00169
SMOVL C00170 +MOVJ EC00170
SMOVL C00171 +MOVJ EC00171
SMOVL C00172 +MOVJ EC00172
SMOVL C00173 +MOVJ EC00173
SMOVL C00174 +MOVJ EC00174
SMOVL C00175 +MOVJ EC00175
SMOVL C00176 +MOVJ EC00176
SMOVL C00177 +MOVJ EC00177
SMOVL C00178 +MOVJ EC00178
SMOVL C00179 +MOVJ EC00179
SMOVL C00180 +MOVJ EC00180
SMOVL C00181 +MOVJ EC00181
SMOVL C00182 +MOVJ EC00182
SMOVL C00183 +MOVJ EC00183
SMOVL C00184 +MOVJ EC00184
SMOVL C00185 +MOVJ EC00185
SMOVL C00186 +MOVJ EC00186
SMOVL C00187 +MOVJ EC00187
SMOVL C00188 +MOVJ EC00188
SMOVL C00189 +MOVJ EC00189
SMOVL C00190 +MOVJ EC00190
SMOVL C00191 +MOVJ EC00191
SMOVL C00192 +MOVJ EC00192
SMOVL C00193 +MOVJ EC00193
SMOVL C00194 +MOVJ EC00194
SMOVL C00195 +MOVJ EC00195
SMOVL C00196 +MOVJ EC00196
SMOVL C00197 +MOVJ EC00197
SMOVL C00198 +MOVJ EC00198
SMOVL C00199 +MOVJ EC00199
SMOVL C00200 +MOVJ EC00200
SMOVL C00201 +MOVJ EC00201
SMOVL C00202 +MOVJ EC00202
SMOVL C00203 +MOVJ EC00203
SMOVL C00204 +MOVJ EC00204
SMOVL C00205 +MOVJ EC00205
SMOVL C00206 +MOVJ EC00206
SMOVL C00207 +MOVJ EC00207
SMOVL C00208 +MOVJ EC00208
SMOVL C00209 +MOVJ EC00209
SMOVL C00210 +MOVJ EC00210
SMOVL C00211 +MOVJ EC00211
SMOVL C00212 +MOVJ EC00212
SMOVL C00213 +MOVJ EC00213
SMOVL C00214 +MOVJ EC00214
SMOVL C00215 +MOVJ EC00215
SMOVL C00216 +MOVJ EC00216
SMOVL C00217 +MOVJ EC00217
SMOVL C00218 +MOVJ EC00218
SMOVL C00219 +MOVJ EC00219
SMOVL C00220 +MOVJ EC00220
SMOVL C00221 +MOVJ EC00221
SMOVL C00222 +MOVJ EC00222
SMOVL C00223 +MOVJ EC00223
SMOVL C00224 +MOVJ EC00224
SMOVL C00225 +MOVJ EC00225
SMOVL C00226 +MOVJ EC00226
SMOVL C00227 +MOVJ EC00227
SMOVL C00228 +MOVJ EC00228
SMOVL C00229 +MOVJ EC00229
SMOVL C00230 +MOVJ EC00230
SMOVL C00231 +MOVJ EC00231
SMOVL C00232 +MOVJ EC00232
SMOVL C00233 +MOVJ EC00233
SMOVL C00234 +MOVJ EC00234
SMOVL C00235 +MOVJ EC00235
SMOVL C00236 +MOVJ EC00236
SMOVL C00237 +MOVJ EC00237
SMOVL C00238 +MOVJ EC00238
SMOVL C00239 +MOVJ EC00239
SMOVL C00240 +MOVJ EC00240
SMOVL C00241 +MOVJ EC00241
SMOVL C00242 +MOVJ EC00242
SMOVL C00243 +MOVJ EC00243
SMOVL C00244 +MOVJ EC00244
SMOVL C00245 +MOVJ EC00245
SMOVL C00246 +MOVJ EC00246
SMOVL C00247 +MOVJ EC00247
SMOVL C00248 +MOVJ EC00248
SMOVL C00249 +MOVJ EC00249
SMOVL C00250 +MOVJ EC00250
SMOVL C00251 +MOVJ EC00251
SMOVL C00252 +MOVJ EC00252
SMOVL C00253 +MOVJ EC00253
SMOVL C00254 +MOVJ EC00254
SMOVL C00255 +MOVJ EC00255
SMOVL C00256 +MOVJ EC00256
SMOVL C00257 +MOVJ EC00257
SMOVL C00258 +MOVJ EC00258
SMOVL C00259 +MOVJ EC00259
SMOVL C00260 +MOVJ EC00260
SMOVL C00261 +MOVJ EC00261
SMOVL C00262 +MOVJ EC00262
SMOVL C00263 +MOVJ EC00263
SMOVL C00264 +MOVJ EC00264
SMOVL C00265 +MOVJ EC00265
SMOVL C00266 +MOVJ EC00266
SMOVL C00267 +MOVJ EC00267
SMOVL C00268 +MOVJ EC00268
SMOVL C00269 +MOVJ EC00269
SMOVL C00270 +MOVJ EC00270
SMOVL C00271 +MOVJ EC00271
SMOVL C00272 +MOVJ EC00272
SMOVL C00273 +MOVJ EC00273
SMOVL C00274 +MOVJ EC00274
SMOVL C00275 +MOVJ EC00275
SMOVL C00276 +MOVJ EC00276
SMOVL C00277 +MOVJ EC00277
SMOVL C00278 +MOVJ EC00278
SMOVL C00279 +MOVJ EC00279
SMOVL C00280 +MOVJ EC00280
SMOVL C00281 +MOVJ EC00281
SMOVL C00282 +MOVJ EC00282
SMOVL C00283 +MOVJ EC00283
SMOVL C00284 +MOVJ EC00284
SMOVL C00285 +MOVJ EC00285
SMOVL C00286 +MOVJ EC00286
SMOVL C00287 +MOVJ EC00287
SMOVL C00288 +MOVJ EC00288
SMOVL C00289 +MOVJ EC00289
SMOVL C00290 +MOVJ EC00290
SMOVL C00291 +MOVJ EC00291
SMOVL C00292 +MOVJ EC00292
SMOVL C00293 +MOVJ EC00293
SMOVL C00294 +MOVJ EC00294
SMOVL C00295 +MOVJ EC00295
SMOVL C00296 +MOVJ EC00296
SMOVL C00297 +MOVJ EC00297
SMOVL C00298 +MOVJ EC00298
SMOVL C00299 +MOVJ EC00299
SMOVL C00300 +MOVJ EC00300
SMOVL C00301 +MOVJ EC00301
SMOVL C00302 +MOVJ EC00302
SMOVL C00303 +MOVJ EC00303
SMOVL C00304 +MOVJ EC00304
SMOVL C00305 +MOVJ EC00305
SMOVL C00306 +MOVJ EC00306
SMOVL C00307 +MOVJ EC00307
SMOVL C00308 +MOVJ EC00308
SMOVL C00309 +MOVJ EC00309
SMOVL C00310 +MOVJ EC00310
SMOVL C00311 +MOVJ EC00311
SMOVL C00312 +MOVJ EC00312
SMOVL C00313 +MOVJ EC00313
SMOVL C00314 +MOVJ EC00314
SMOVL C00315 +MOVJ EC00315
SMOVL C00316 +MOVJ EC00316
SMOVL C00317 +MOVJ EC00317
SMOVL C00318 +MOVJ EC00318
SMOVL C00319 +MOVJ EC00319
SMOVL C00320 +MOVJ EC00320
SMOVL C00321 +MOVJ EC00321
SMOVL C00322 +MOVJ EC00322
SMOVL C00323 +MOVJ EC00323
SMOVL C00324 +MOVJ EC00324
SMOVL C00325 +MOVJ EC00325
SMOVL C00326 +MOVJ EC00326
SMOVL C00327 +MOVJ EC00327
SMOVL C00328 +MOVJ EC00328
SMOVL C00329 +MOVJ EC00329
SMOVL C00330 +MOVJ EC00330
SMOVL C00331 +MOVJ EC00331
SMOVL C00332 +MOVJ EC00332
SMOVL C00333 +MOVJ EC00333
SMOVL C00334 +MOVJ EC00334
SMOVL C00335 +MOVJ EC00335
SMOVL C00336 +MOVJ EC00336
SMOVL C00337 +MOVJ EC00337
SMOVL C00338 +MOVJ EC00338
SMOVL C00339 +MOVJ EC00339
SMOVL C00340 +MOVJ EC00340
SMOVL C00341 +MOVJ EC00341
SMOVL C00342 +MOVJ EC00342
SMOVL C00343 +MOVJ EC00343
SMOVL C00344 +MOVJ EC00344
SMOVL C00345 +MOVJ EC00345
SMOVL C00346 +MOVJ EC00346
SMOVL C00347 +MOVJ EC00347
SMOVL C00348 +MOVJ EC00348
SMOVL C00349 +MOVJ EC00349
SMOVL C00350 +MOVJ EC00350
SMOVL C00351 +MOVJ EC00351
SMOVL C00352 +MOVJ EC00352
SMOVL C00353 +MOVJ EC00353
SMOVL C00354 +MOVJ EC00354
SMOVL C00355 +MOVJ EC00355
SMOVL C00356 +MOVJ EC00356
SMOVL C00357 +MOVJ EC00357
SMOVL C00358 +MOVJ EC00358
SMOVL C00359 +MOVJ EC00359
SMOVL C00360 +MOVJ EC00360
SMOVL C00361 +MOVJ EC00361
SMOVL C00362 +MOVJ EC00362
SMOVL C00363 +MOVJ EC00363
SMOVL C00364 +MOVJ EC00364
SMOVL C00365 +MOVJ EC00365
SMOVL C00366 +MOVJ EC00366
SMOVL C00367 +MOVJ EC00367
SMOVL C00368 +MOVJ EC00368
SMOVL C00369 +MOVJ EC00369
SMOVL C00370 +MOVJ EC00370
SMOVL C00371 +MOVJ EC00371
SMOVL C00372 +MOVJ EC00372
SMOVL C00373 +MOVJ EC00373
SMOVL C00374 +MOVJ EC00374
SMOVL C00375 +MOVJ EC00375
SMOVL C00376 +MOVJ EC00376
SMOVL C00377 +MOVJ EC00377
SMOVL C00378 +MOVJ EC00378
SMOVL C00379 +MOVJ EC00379
SMOVL C00380 +MOVJ EC00380
SMOVL C00381 +MOVJ EC00381
SMOVL C00382 +MOVJ EC00382
SMOVL C00383 +MOVJ EC00383
SMOVL C00384 +MOVJ EC00384
SMOVL C00385 +MOVJ EC00385
SMOVL C00386 +MOVJ EC00386
SMOVL C00387 +MOVJ EC00387
SMOVL C00388 +MOVJ EC00388
SMOVL C00389 +MOVJ EC00389
SMOVL C00390 +MOVJ EC00390
SMOVL C00391 +MOVJ EC00391
SMOVL C00392 +MOVJ EC00392
SMOVL C00393 +MOVJ EC00393
SMOVL C00394 +MOVJ EC00394
SMOVL C00395 +MOVJ EC00395
SMOVL C00396 +MOVJ EC00396
SMOVL C00397 +MOVJ EC00397
SMOVL C00398 +MOVJ EC00398
SMOVL C00399 +MOVJ EC00399
SMOVL C00400 +MOVJ EC00400
SMOVL C00401 +MOVJ EC00401
SMOVL C00402 +MOVJ EC00402
SMOVL C00403 +MOVJ EC00403
SMOVL C00404 +MOVJ EC00404
SMOVL C00405 +MOVJ EC00405
SMOVL C00406 +MOVJ EC00406
SMOVL C00407 +MOVJ EC00407
SMOVL C00408 +MOVJ EC00408
SMOVL C00409 +MOVJ EC00409
SMOVL C00410 +MOVJ EC00410
SMOVL C00411 +MOVJ EC00411
SMOVL C00412 +MOVJ EC00412
SMOVL C00413 +MOVJ EC00413
SMOVL C00414 +MOVJ EC00414
SMOVL C00415 +MOVJ EC00415
SMOVL C00416 +MOVJ EC00416
SMOVL C00417 +MOVJ EC00417
SMOVL C00418 +MOVJ EC00418
SMOVL C00419 +MOVJ EC00419
SMOVL C00420 +MOVJ EC00420
SMOVL C00421 +MOVJ EC00421
SMOVL C00422 +MOVJ EC00422
SMOVL C00423 +MOVJ EC00423
SMOVL C00424 +MOVJ EC00424
SMOVL C00425 +MOVJ EC00425
SMOVL C00426 +MOVJ EC00426
SMOVL C00427 +MOVJ EC00427
SMOVL C00428 +MOVJ EC00428
SMOVL C00429 +MOVJ EC00429
SMOVL C00430 +MOVJ EC00430
SMOVL C00431 +MOVJ EC00431
SMOVL C00432 +MOVJ EC00432
SMOVL C00433 +MOVJ EC00433
SMOVL C00434 +MOVJ EC00434
SMOVL C00435 +MOVJ EC00435
SMOVL C00436 +MOVJ EC00436
SMOVL C00437 +MOVJ EC00437
SMOVL C00438 +MOVJ EC00438
SMOVL C00439 +MOVJ EC00439
SMOVL C00440 +MOVJ EC00440
SMOVL C00441 +MOVJ EC00441
SMOVL C00442 +MOVJ EC00442
SMOVL C00443 +MOVJ EC00443
SMOVL C00444 +MOVJ EC00444
SMOVL C00445 +MOVJ EC00445
SMOVL C00446 +MOVJ EC00446
SMOVL C00447 +MOVJ EC00447
SMOVL C00448 +MOVJ EC00448
SMOVL C00449 +MOVJ EC00449
SMOVL C00450 +MOVJ EC00450
SMOVL C00451 +MOVJ EC00451
SMOVL C00452 +MOVJ EC00452
SMOVL C00453 +MOVJ EC00453
SMOVL C00454 +MOVJ EC00454
SMOVL C00455 +MOVJ EC00455
SMOVL C00456 +MOVJ EC00456
SMOVL C00457 +MOVJ EC00457
SMOVL C00458 +MOVJ EC00458
SMOVL C00459 +MOVJ EC00459
SMOVL C00460 +MOVJ EC00460
SMOVL C00461 +MOVJ EC00461
SMOVL C00462 +MOVJ EC00462
SMOVL C00463 +MOVJ EC00463
SMOVL C00464 +MOVJ EC00464
SMOVL C00465 +MOVJ EC00465
SMOVL C00466 +MOVJ EC00466
SMOVL C00467 +MOVJ EC00467
SMOVL C00468 +MOVJ EC00468
SMOVL C00469 +MOVJ EC00469
SMOVL C00470 +MOVJ EC00470
SMOVL C00471 +MOVJ EC00471
SMOVL C00472 +MOVJ EC00472
SMOVL C00473 +MOVJ EC00473
SMOVL C00474 +MOVJ EC00474
SMOVL C00475 +MOVJ EC00475
SMOVL C00476 +MOVJ EC00476
SMOVL C00477 +MOVJ EC00477
SMOVL C00478 +MOVJ EC00478
SMOVL C00479 +MOVJ EC00479
SMOVL C00480 +MOVJ EC00480
SMOVL C00481 +MOVJ EC00481
SMOVL C00482 +MOVJ EC00482
SMOVL C00483 +MOVJ EC00483
SMOVL C00484 +MOVJ EC00484
SMOVL C00485 +MOVJ EC00485
SMOVL C00486 +MOVJ EC00486
SMOVL C00487 +MOVJ EC00487
SMOVL C00488 +MOVJ EC00488
SMOVL C00489 +MOVJ EC00489
SMOVL C00490 +MOVJ EC00490
SMOVL C00491 +MOVJ EC00491
SMOVL C00492 +MOVJ EC00492
SMOVL C00493 +MOVJ EC00493
SMOVL C00494 +MOVJ EC00494
SMOVL C00495 +MOVJ EC00495
SMOVL C00496 +MOVJ EC00496
SMOVL C00497 +MOVJ EC00497
SMOVL C00498 +MOVJ EC00498
SMOVL C00499 +MOVJ EC00499
SMOVL C00500 +MOVJ EC00500
SMOVL C00501 +MOVJ EC00501
SMOVL C00502 +MOVJ EC00502
SMOVL C00503 +MOVJ EC00503
SMOVL C00504 +MOVJ EC00504
SMOVL C00505 +MOVJ EC00505
SMOVL C00506 +MOVJ EC00506
SMOVL C00507 +MOVJ EC00507
SMOVL C00508 +MOVJ EC00508
SMOVL C00509 +MOVJ EC00509
SMOVL C00510 +MOVJ EC00510
SMOVL C00511 +MOVJ EC00511
SMOVL C00512 +MOVJ EC00512
SMOVL C00513 +MOVJ EC00513
SMOVL C00514 +MOVJ EC00514
SMOVL C00515 +MOVJ EC00515
SMOVL C00516 +MOVJ EC00516
SMOVL C00517 +MOVJ EC00517
SMOVL C00518 +MOVJ EC00518
SMOVL C00519 +MOVJ EC00519
SMOVL C00520 +MOVJ EC00520
SMOVL C00521 +MOVJ EC00521
SMOVL C00522 +MOVJ EC00522
SMOVL C00523 +MOVJ EC00523
SMOVL C00524 +MOVJ EC00524
SMOVL C00525 +MOVJ EC00525
SMOVL C00526 +MOVJ EC00526
SMOVL C00527 +MOVJ EC00527
SMOVL C00528 +MOVJ EC00528
SMOVL C00529 +MOVJ EC00529
SMOVL C00530 +MOVJ EC00530
SMOVL C00531 +MOVJ EC00531
SMOVL C00532 +MOVJ EC00532
SMOVL C00533 +MOVJ EC00533
SMOVL C00534 +MOVJ EC00534
SMOVL C00535 +MOVJ EC00535
SMOVL C00536 +MOVJ EC00536
SMOVL C00537 +MOVJ EC00537
SMOVL C00538 +MOVJ EC00538
SMOVL C00539 +MOVJ EC00539
SMOVL C00540 +MOVJ EC00540
SMOVL C00541 +MOVJ EC00541
SMOVL C00542 +MOVJ EC00542
SMOVL C00543 +MOVJ EC00543
SMOVL C00544 +MOVJ EC00544
SMOVL C00545 +MOVJ EC00545
SMOVL C00546 +MOVJ EC00546
SMOVL C00547 +MOVJ EC00547
SMOVL C00548 +MOVJ EC00548
SMOVL C00549 +MOVJ EC00549
SMOVL C00550 +MOVJ EC00550
SMOVL C00551 +MOVJ EC00551
SMOVL C00552 +MOVJ EC00552
SMOVL C00553 +MOVJ EC00553
SMOVL C00554 +MOVJ EC00554
SMOVL C00555 +MOVJ EC00555
SMOVL C00556 +MOVJ EC00556
SMOVL C00557 +MOVJ EC00557
SMOVL C00558 +MOVJ EC00558
SMOVL C00559 +MOVJ EC00559
SMOVL C00560 +MOVJ EC00560
SMOVL C00561 +MOVJ EC00561
SMOVL C00562 +MOVJ EC00562
SMOVL C00563 +MOVJ EC00563
SMOVL C00564 +MOVJ EC00564
SMOVL C00565 +MOVJ EC00565
SMOVL C00566 +MOVJ EC00566
SMOVL C00567 +MOVJ EC00567
SMOVL C00568 +MOVJ EC00568
SMOVL C00569 +MOVJ EC00569
SMOVL C00570 +MOVJ EC00570
SMOVL C00571 +MOVJ EC00571
SMOVL C00572 +MOVJ EC00572
SMOVL C00573 +MOVJ EC00573
SMOVL C00574 +MOVJ EC00574
SMOVL C00575 +MOVJ EC00575
SMOVL C00576 +MOVJ EC00576
SMOVL C00577 +MOVJ EC00577
SMOVL C00578 +MOVJ EC00578
SMOVL C00579 +MOVJ EC00579
SMOVL C00580 +MOVJ EC00580
SMOVL C00581 +MOVJ EC00581
SMOVL C00582 +MOVJ EC00582
SMOVL C00583 +MOVJ EC00583
SMOVL C00584 +MOVJ EC00584
SMOVL C00585 +MOVJ EC00585
SMOVL C00586 +MOVJ EC00586
SMOVL C00587 +MOVJ EC00587
SMOVL C00588 +MOVJ EC00588
SMOVL C00589 +MOVJ EC00589
SMOVL C00590 +MOVJ EC00590
SMOVL C00591 +MOVJ EC00591
SMOVL C00592 +MOVJ EC00592
SMOVL C00593 +MOVJ EC00593
SMOVL C00594 +MOVJ EC00594
SMOVL C00595 +MOVJ EC00595
SMOVL C00596 +MOVJ EC00596
SMOVL C00597 +MOVJ EC00597
SMOVL C00598 +MOVJ EC00598
SMOVL C00599 +MOVJ EC00599
SMOVL C00600 +MOVJ EC00600
SMOVL C00601 +MOVJ EC00601
SMOVL C00602 +MOVJ EC00602
SMOVL C00603 +MOVJ EC00603
SMOVL C00604 +MOVJ EC00604
SMOVL C00605 +MOVJ EC00605
SMOVL C00606 +MOVJ EC00606
SMOVL C00607 +MOVJ EC00607
SMOVL C00608 +MOVJ EC00608
SMOVL C00609 +MOVJ EC00609
SMOVL C00610 +MOVJ EC00610
SMOVL C00611 +MOVJ EC00611
SMOVL C00612 +MOVJ EC00612
SMOVL C00613 +MOVJ EC00613
SMOVL C00614 +MOVJ EC00614
SMOVL C00615 +MOVJ EC00615
SMOVL C00616 +MOVJ EC00616
SMOVL C00617 +MOVJ EC00617
SMOVL C00618 +MOVJ EC00618
SMOVL C00619 +MOVJ EC00619
SMOVL C00620 +MOVJ EC00620
SMOVL C00621 +MOVJ EC00621
SMOVL C00622 +MOVJ EC00622
SMOVL C00623 +MOVJ EC00623
SMOVL C00624 +MOVJ EC00624
SMOVL C00625 +MOVJ EC00625
SMOVL C00626 +MOVJ EC00626
SMOVL C00627 +MOVJ EC00627
SMOVL C00628 +MOVJ EC00628
SMOVL C00629 +MOVJ EC00629
SMOVL C00630 +MOVJ EC00630
SMOVL C00631 +MOVJ EC00631
SMOVL C00632 +MOVJ EC00632
SMOVL C00633 +MOVJ EC00633
SMOVL C00634 +MOVJ EC00634
SMOVL C00635 +MOVJ EC00635
SMOVL C00636 +MOVJ EC00636
SMOVL C00637 +MOVJ EC00637
SMOVL C00638 +MOVJ EC00638
SMOVL C00639 +MOVJ EC00639
SMOVL C00640 +MOVJ EC00640
SMOVL C00641 +MOVJ EC00641
SMOVL C00642 +MOVJ EC00642
SMOVL C00643 +MOVJ EC00643
SMOVL C00644 +MOVJ EC00644
SMOVL C00645 +MOVJ EC00645
SMOVL C00646 +MOVJ EC00646
SMOVL C00647 +MOVJ EC00647
SMOVL C00648 +MOVJ EC00648
SMOVL C00649 +MOVJ EC00649
SMOVL C00650 +MOVJ EC00650
SMOVL C00651 +MOVJ EC00651
SMOVL C00652 +MOVJ EC00652
SMOVL C00653 +MOVJ EC00653
SMOVL C00654 +MOVJ EC00654
SMOVL C00655 +MOVJ EC00655
SMOVL C00656 +MOVJ EC00656
SMOVL C00657 +MOVJ EC00657
SMOVL C00658 +MOVJ EC00658
SMOVL C00659 +MOVJ EC00659
SMOVL C00660 +MOVJ EC00660
SMOVL C00661 +MOVJ EC00661
SMOVL C00662 +MOVJ EC00662
SMOVL C00663 +MOVJ EC00663
SMOVL C00664 +MOVJ EC00664
SMOVL C00665 +MOVJ EC00665
SMOVL C00666 +MOVJ EC00666
SMOVL C00667 +MOVJ EC00667
SMOVL C00668 +MOVJ EC00668
SMOVL C00669 +MOVJ EC00669
SMOVL C00670 +MOVJ EC00670
SMOVL C00671 +MOVJ EC00671
SMOVL C00672 +MOVJ EC00672
SMOVL C00673 +MOVJ EC00673
SMOVL C00674 +MOVJ EC00674
SMOVL C00675 +MOVJ EC00675
SMOVL C00676 +MOVJ EC00676
SMOVL C00677 +MOVJ EC00677
SMOVL C00678 +MOVJ EC00678
SMOVL C00679 +MOVJ EC00679
SMOVL C00680 +MOVJ EC00680
SMOVL C00681 +MOVJ EC00681
SMOVL C00682 +MOVJ EC00682
SMOVL C00683 +MOVJ EC00683
SMOVL C00684 +MOVJ EC00684
SMOVL C00685 +MOVJ EC00685
SMOVL C00686 +MOVJ EC00686
SMOVL C00687 +MOVJ EC00687
SMOVL C00688 +MOVJ EC00688
SMOVL C00689 +MOVJ EC00689
SMOVL C00690 +MOVJ EC00690
SMOVL C00691 +MOVJ EC00691
SMOVL C00692 +MOVJ EC00692
SMOVL C00693 +MOVJ EC00693
SMOVL C00694 +MOVJ EC00694
SMOVL C00695 +MOVJ EC00695
SMOVL C00696 +MOVJ EC00696
SMOVL C00697 +MOVJ EC00697
SMOVL C00698 +MOVJ EC00698
SMOVL C00699 +MOVJ EC00699
SMOVL C00700 +MOVJ EC00700
SMOVL C00701 +MOVJ EC00701
SMOVL C00702 +MOVJ EC00702
SMOVL C00703 +MOVJ EC00703
SMOVL C00704 +MOVJ EC00704
SMOVL C00705 +MOVJ EC00705
SMOVL C00706 +MOVJ EC00706
SMOVL C00707 +MOVJ EC00707
SMOVL C00708 +MOVJ EC00708
SMOVL C00709 +MOVJ EC00709
SMOVL C00710 +MOVJ EC00710
SMOVL C00711 +MOVJ EC00711
SMOVL C00712 +MOVJ EC00712
SMOVL C00713 +MOVJ EC00713
SMOVL C00714 +MOVJ EC00714
SMOVL C00715 +MOVJ EC00715
SMOVL C00716 +MOVJ EC00716
SMOVL C00717 +MOVJ EC00717
SMOVL C00718 +MOVJ EC00718
SMOVL C00719 +MOVJ EC00719
SMOVL C00720 +MOVJ EC00720
SMOVL C00721 +MOVJ EC00721
SMOVL C00722 +MOVJ EC00722
SMOVL C00723 +MOVJ EC00723
SMOVL C00724 +MOVJ EC00724
SMOVL C00725 +MOVJ EC00725
SMOVL C00726 +MOVJ EC00726
SMOVL C00727 +MOVJ EC00727
SMOVL C00728 +MOVJ EC00728
SMOVL C00729 +MOVJ EC00729
SMOVL C00730 +MOVJ EC00730
SMOVL C00731 +MOVJ EC00731
SMOVL C00732 +MOVJ EC00732
SMOVL C00733 +MOVJ EC00733
SMOVL C00734 +MOVJ EC00734
SMOVL C00735 +MOVJ EC00735
SMOVL C00736 +MOVJ EC00736
SMOVL C00737 +MOVJ EC00737
SMOVL C00738 +MOVJ EC00738
SMOVL C00739 +MOVJ EC00739
SMOVL C00740 +MOVJ EC00740
SMOVL C00741 +MOVJ EC00741
SMOVL C00742 +MOVJ EC00742
SMOVL C00743 +MOVJ EC00743
SMOVL C00744 +MOVJ EC00744
SMOVL C00745 +MOVJ EC00745
SMOVL C00746 +MOVJ EC00746
SMOVL C00747 +MOVJ EC00747
SMOVL C00748 +MOVJ EC00748
SMOVL C00749 +MOVJ EC00749
SMOVL C00750 +MOVJ EC00750
SMOVL C00751 +MOVJ EC00751
SMOVL C00752 +MOVJ EC00752
SMOVL C00753 +MOVJ EC00753
SMOVL C00754 +MOVJ EC00754
SMOVL C00755 +MOVJ EC00755
SMOVL C00756 +MOVJ EC00756
SMOVL C00757 +MOVJ EC00757
SMOVL C00758 +MOVJ EC00758
SMOVL C00759 +MOVJ EC00759
SMOVL C00760 +MOVJ EC00760
SMOVL C00761 +MOVJ EC00761
SMOVL C00762 +MOVJ EC00762
SMOVL C00763 +MOVJ EC00763
SMOVL C00764 +MOVJ EC00764
SMOVL C00765 +MOVJ EC00765
SMOVL C00766 +MOVJ EC00766
SMOVL C00767 +MOVJ EC00767
SMOVL C00768 +MOVJ EC00768
SMOVL C00769 +MOVJ EC00769
SMOVL C00770 +MOVJ EC00770
SMOVL C00771 +MOVJ EC00771
SMOVL C00772 +MOVJ EC00772
SMOVL C00773 +MOVJ EC00773
SMOVL C00774 +MOVJ EC00774
SMOVL C00775 +MOVJ EC00775
SMOVL C00776 +MOVJ EC00776
SMOVL C00777 +MOVJ EC00777
SMOVL C00778 +MOVJ EC00778
SMOVL C00779 +MOVJ EC00779
SMOVL C00780 +MOVJ EC00780
SMOVL C00781 +MOVJ EC00781
SMOVL C00782 +MOVJ EC00782
SMOVL C00783 +MOVJ EC00783
SMOVL C00784 +MOVJ EC00784
SMOVL C00785 +MOVJ EC00785
SMOVL C00786 +MOVJ EC00786
SMOVL C00787 +MOVJ EC00787
SMOVL C00788 +MOVJ EC00788
SMOVL C00789 +MOVJ EC00789
SMOVL C00790 +MOVJ EC00790
SMOVL C00791 +MOVJ EC00791
SMOVL C00792 +MOVJ EC00792
SMOVL C00793 +MOVJ EC00793
SMOVL C00794 +MOVJ EC00794
SMOVL C00795 +MOVJ EC00795
SMOVL C00796 +MOVJ EC00796
SMOVL C00797 +MOVJ EC00797
SMOVL C00798 +MOVJ EC00798
SMOVL C00799 +MOVJ EC00799
SMOVL C00800 +MOVJ EC00800
SMOVL C00801 +MOVJ EC00801
SMOVL C00802 +MOVJ EC00802
SMOVL C00803 +MOVJ EC00803
SMOVL C00804 +MOVJ EC00804
SMOVL C00805 +MOVJ EC00805
SMOVL C00806 +MOVJ EC00806
SMOVL C00807 +MOVJ EC00807
SMOVL C00808 +MOVJ EC00808
SMOVL C00809 +MOVJ EC00809
SMOVL C00810 +MOVJ EC00810
SMOVL C00811 +MOVJ EC00811
SMOVL C00812 +MOVJ EC00812
SMOVL C00813 +MOVJ EC00813
SMOVL C00814 +MOVJ EC00814
SMOVL C00815 +MOVJ EC00815
SMOVL C00816 +MOVJ EC00816
SMOVL C00817 +MOVJ EC00817
SMOVL C00818 +MOVJ EC00818
SMOVL C00819 +MOVJ EC00819
SMOVL C00820 +MOVJ EC00820
SMOVL C00821 +MOVJ EC00821
SMOVL C00822 +MOVJ EC00822
SMOVL C00823 +MOVJ EC00823
SMOVL C00824 +MOVJ EC00824
SMOVL C00825 +MOVJ EC00825
SMOVL C00826 +MOVJ EC00826
SMOVL C00827 +MOVJ EC00827
SMOVL C00828 +MOVJ EC00828
SMOVL C00829 +MOVJ EC00829
SMOVL C00830 +MOVJ EC00830
SMOVL C00831 +MOVJ EC00831
SMOVL C00832 +MOVJ EC00832
SMOVL C00833 +MOVJ EC00833
SMOVL C00834 +MOVJ EC00834
SMOVL C00835 +MOVJ EC00835
SMOVL C00836 +MOVJ EC00836
SMOVL C00837 +MOVJ EC00837
SMOVL C00838 +MOVJ EC00838
SMOVL C00839 +MOVJ EC00839
SMOVL C00840 +MOVJ EC00840
SMOVL C00841 +MOVJ EC00841
SMOVL C00842 +MOVJ EC00842
SMOVL C00843 +MOVJ EC00843
SMOVL C00844 +MOVJ EC00844
SMOVL C00845 +MOVJ EC00845
SMOVL C00846 +MOVJ EC00846
SMOVL C00847 +MOVJ EC00847
SMOVL C00848 +MOVJ EC00848
SMOVL C00849 +MOVJ EC00849
SMOVL C00850 +MOVJ EC00850
SMOVL C00851 +MOVJ EC00851
SMOVL C00852 +MOVJ EC00852
SMOVL C00853 +MOVJ EC00853
SMOVL C00854 +MOVJ EC00854
SMOVL C00855 +MOVJ EC00855
SMOVL C00856 +MOVJ EC00856
SMOVL C00857 +MOVJ EC00857
SMOVL C00858 +MOVJ EC00858
SMOVL C00859 +MOVJ EC00859
SMOVL C00860 +MOVJ EC00860
SMOVL C00861 +MOVJ EC00861
SMOVL C00862 +MOVJ EC00862
SMOVL C00863 +MOVJ EC00863
SMOVL C00864 +MOVJ EC00864
SMOVL C00865 +MOVJ EC00865
SMOVL C00866 +MOVJ EC00866
SMOVL C00867 +MOVJ EC00867
SMOVL C00868 +MOVJ EC00868
SMOVL C00869 +MOVJ EC00869
SMOVL C00870 +MOVJ EC00870
SMOVL C00871 +MOVJ EC00871
SMOVL C00872 +MOVJ EC00872
SMOVL C00873 +MOVJ EC00873
SMOVL C00874 +MOVJ EC00874
SMOVL C00875 +MOVJ EC00875
SMOVL C00876 +MOVJ EC00876
SMOVL C00877 +MOVJ EC00877
SMOVL C00878 +MOVJ EC00878
SMOVL C00879 +MOVJ EC00879
SMOVL C00880 +MOVJ EC00880
SMOVL C00881 +MOVJ EC00881
SMOVL C00882 +MOVJ EC00882
SMOVL C00883 +MOVJ EC00883
SMOVL C00884 +MOVJ EC00884
SMOVL C00885 +MOVJ EC00885
SMOVL C00886 +MOVJ EC00886
SMOVL C00887 +MOVJ EC00887
SMOVL C00888 +MOVJ EC00888
SMOVL C00889 +MOVJ EC00889
SMOVL C00890 +MOVJ EC00890
SMOVL C00891 +MOVJ EC00891
SMOVL C00892 +MOVJ EC00892
SMOVL C00893 +MOVJ EC00893
SMOVL C00894 +MOVJ EC00894
SMOVL C00895 +MOVJ EC00895
SMOVL C00896 +MOVJ EC00896
SMOVL C00897 +MOVJ EC00897
SMOVL C00898 +MOVJ EC00898
SMOVL C00899 +MOVJ EC00899
SMOVL C00900 +MOVJ EC00900
SMOVL C00901 +MOVJ EC00901
SMOVL C00902 +MOVJ EC00902
SMOVL C00903 +MOVJ EC00903
SMOVL C00904 +MOVJ EC00904
SMOVL C00905 +MOVJ EC00905
SMOVL C00906 +MOVJ EC00906
SMOVL C00907 +MOVJ EC00907
SMOVL C00908 +MOVJ EC00908
SMOVL C00909 +MOVJ EC00909
SMOVL C00910 +MOVJ EC00910
SMOVL C00911 +MOVJ EC00911
SMOVL C00912 +MOVJ EC00912
SMOVL C00913 +MOVJ EC00913
SMOVL C00914 +MOVJ EC00914
SMOVL C00915 +MOVJ EC00915
SMOVL C00916 +MOVJ EC00916
SMOVL C00917 +MOVJ EC00917
SMOVL C00918 +MOVJ EC00918
SMOVL C00919 +MOVJ EC00919
SMOVL C00920 +MOVJ EC00920
SMOVL C00921 +MOVJ EC00921
SMOVL C00922 +MOVJ EC00922
SMOVL C00923 +MOVJ EC00923
SMOVL C00924 +MOVJ EC00924
SMOVL C00925 +MOVJ EC00925
SMOVL C00926 +MOVJ EC00926
SMOVL C00927 +MOVJ EC00927
SMOVL C00928 +MOVJ EC00928
SMOVL C00929 +MOVJ EC00929
SMOVL C00930 +MOVJ EC00930
SMOVL C00931 +MOVJ EC00931
SMOVL C00932 +MOVJ EC00932
SMOVL C00933 +MOVJ EC00933
SMOVL C00934 +MOVJ EC00934
SMOVL C00935 +MOVJ EC00935
SMOVL C00936 +MOVJ EC00936
SMOVL C00937 +MOVJ EC00937
SMOVL C00938 +MOVJ EC00938
SMOVL C00939 +MOVJ EC00939
SMOVL C00940 +MOVJ EC00940
SMOVL C00941 +MOVJ EC00941
SMOVL C00942 +MOVJ EC00942
SMOVL C00943 +MOVJ EC00943
SMOVL C00944 +MOVJ EC00944
SMOVL C00945 +MOVJ EC00945
SMOVL C00946 +MOVJ EC00946
SMOVL C00947 +MOVJ EC00947
SMOVL C00948 +MOVJ EC00948
SMOVL C00949 +MOVJ EC00949
SMOVL C00950 +MOVJ EC00950
SMOVL C00951 +MOVJ EC00951
SMOVL C00952 +MOVJ EC00952
SMOVL C00953 +MOVJ EC00953
SMOVL C00954 +MOVJ EC00954
SMOVL C00955 +MOVJ EC00955
SMOVL C00956 +MOVJ EC00956
SMOVL C00957 +MOVJ EC00957
SMOVL C00958 +MOVJ EC00958
SMOVL C00959 +MOVJ EC00959
SMOVL C00960 +MOVJ EC00960
SMOVL C00961 +MOVJ EC00961
SMOVL C00962 +MOVJ EC00962
SMOVL C00963 +MOVJ EC00963
SMOVL C00964 +MOVJ EC00964
SMOVL C00965 +MOVJ EC00965
SMOVL C00966 +MOVJ EC00966
SMOVL C00967 +MOVJ EC00967
SMOVL C00968 +MOVJ EC00968
SMOVL C00969 +MOVJ EC00969
SMOVL C00970 +MOVJ EC00970
SMOVL C00971 +MOVJ EC00971
SMOVL C00972 +MOVJ EC00972
SMOVL C00973 +MOVJ EC00973
SMOVL C00974 +MOVJ EC00974
SMOVL C00975 +MOVJ EC00975
SMOVL C00976 +MOVJ EC00976
SMOVL C00977 +MOVJ EC00977
SMOVL C00978 +MOVJ EC00978
SMOVL C00979 +MOVJ EC00979
SMOVL C00980 +MOVJ EC00980
SMOVL C00981 +MOVJ EC00981
SMOVL C00982 +MOVJ EC00982
SMOVL C00983 +MOVJ EC00983
SMOVL C00984 +MOVJ EC00984
SMOVL C00985 +MOVJ EC00985
SMOVL C00986 +MOVJ EC00986
SMOVL C00987 +MOVJ EC00987
SMOVL C00988 +MOVJ EC00988
SMOVL C00989 +MOVJ EC00989
SMOVL C00990 +MOVJ EC00990
SMOVL C00991 +MOVJ EC00991
SMOVL C00992 +MOVJ EC00992
SMOVL C00993 +MOVJ EC00993
SMOVL C00994 +MOVJ EC00994
SMOVL C00995 +MOVJ EC00995
SMOVL C00996 +MOVJ EC00996
SMOVL C00997 +MOVJ EC00997
SMOVL C00998 +MOVJ EC00998
SMOVL C00999 +MOVJ EC00999
SMOVL C01000 +MOVJ EC01000
SMOVL C01001 +MOVJ EC01001
SMOVL C01002 +MOVJ EC01002
SMOVL C01003 +MOVJ EC01003
SMOVL C01004 +MOVJ EC01004
SMOVL C01005 +MOVJ EC01005
SMOVL C01006 +MOVJ EC01006
SMOVL C01007 +MOVJ EC01007
SMOVL C01008 +MOVJ EC01008
SMOVL C01009 +MOVJ EC01009
SMOVL C01010 +MOVJ EC01010
SMOVL C01011 +MOVJ EC01011
SMOVL C01012 +MOVJ EC01012
SMOVL C01013 +MOVJ EC01013
SMOVL C01014 +MOVJ EC01014
SMOVL C01015 +MOVJ EC01015
SMOVL C01016 +MOVJ EC01016
SMOVL C01017 +MOVJ EC01017
SMOVL C01018 +MOVJ EC01018
SMOVL C01019 +MOVJ EC01019
SMOVL C01020 +MOVJ EC01020
SMOVL C01021 +MOVJ EC01021
SMOVL C01022 +MOVJ EC01022
SMOVL C01023 +MOVJ EC01023
SMOVL C01024 +MOVJ EC01024
SMOVL C01025 +MOVJ EC01025
SMOVL C01026 +MOVJ EC01026
SMOVL C01027 +MOVJ EC01027
SMOVL C01028 +MOVJ EC01028
SMOVL C01029 +MOVJ EC01029
SMOVL C01030 +MOVJ EC01030
SMOVL C01031 +MOVJ EC01031
SMOVL C01032 +MOVJ EC01032
SMOVL C01033 +MOVJ EC01033
SMOVL C01034 +MOVJ EC01034
SMOVL C01035 +MOVJ EC01035
SMOVL C01036 +MOVJ EC01036
SMOVL C01037 +MOVJ EC01037
SMOVL C01038 +MOVJ EC01038
SMOVL C01039 +MOVJ EC01039
SMOVL C01040 +MOVJ EC01040
SMOVL C01041 +MOVJ EC01041
SMOVL C01042 +MOVJ EC01042
SMOVL C01043 +MOVJ EC01043
SMOVL C01044 +MOVJ EC01044
SMOVL C01045 +MOVJ EC01045
SMOVL C01046 +MOVJ EC01046
SMOVL C01047 +MOVJ EC01047
SMOVL C01048 +MOVJ EC01048
SMOVL C01049 +MOVJ EC01049
SMOVL C01050 +MOVJ EC01050
SMOVL C01051 +MOVJ EC01051
SMOVL C01052 +MOVJ EC01052
SMOVL C01053 +MOVJ EC01053
SMOVL C01054 +MOVJ EC01054
SMOVL C01055 +MOVJ EC01055
SMOVL C01056 +MOVJ EC01056
SMOVL C01057 +MOVJ EC01057
SMOVL C01058 +MOVJ EC01058
SMOVL C01059 +MOVJ EC01059
SMOVL C01060 +MOVJ EC01060
SMOVL C01061 +MOVJ EC01061
SMOVL C01062 +MOVJ EC01062
SMOVL C01063 +MOVJ EC01063
SMOVL C01064 +MOVJ EC01064
SMOVL C01065 +MOVJ EC01065
SMOVL C01066 +MOVJ EC01066
SMOVL C01067 +MOVJ EC01067
SMOVL C01068 +MOVJ EC01068
SMOVL C01069 +MOVJ EC01069
SMOVL C01070 +MOVJ EC01070
SMOVL C01071 +MOVJ EC01071
SMOVL C01072 +MOVJ EC01072
SMOVL C01073 +MOVJ EC01073
SMOVL C01074 +MOVJ EC01074
SMOVL C01075 +MOVJ EC01075
SMOVL C01076 +MOVJ EC01076
SMOVL C01077 +MOVJ EC01077
SMOVL C01078 +MOVJ EC01078
SMOVL C01079 +MOVJ EC01079
SMOVL C01080 +MOVJ EC01080
SMOVL C01081 +MOVJ EC01081
SMOVL C01082 +MOVJ EC01082
SMOVL C01083 +MOVJ EC01083
SMOVL C01084 +MOVJ EC01084
SMOVL C01085 +MOVJ EC01085
SMOVL C01086 +MOVJ EC01086
SMOVL C01087 +MOVJ EC01087
SMOVL C01088 +MOVJ EC01088
SMOVL C01089 +MOVJ EC01089
SMOVL C01090 +MOVJ EC01090
SMOVL C01091 +MOVJ EC01091
SMOVL C01092 +MOVJ EC01092
SMOVL C01093 +MOVJ EC01093
SMOVL C01094 +MOVJ EC01094
SMOVL C01095 +MOVJ EC01095
SMOVL C01096 +MOVJ EC01096
SMOVL C01097 +MOVJ EC01097
SMOVL C01098 +MOVJ EC01098
SMOVL C01099 +MOVJ EC01099
SMOVL C01100 +MOVJ EC01100
SMOVL C01101 +MOVJ EC01101
SMOVL C01102 +MOVJ EC01102
SMOVL C01103 +MOVJ EC01103
SMOVL C01104 +MOVJ EC01104
SMOVL C01105 +MOVJ EC01105
SMOVL C01106 +MOVJ EC01106
SMOVL C01107 +MOVJ EC01107
SMOVL C01108 +MOVJ EC01108
SMOVL C01109 +MOVJ EC01109
SMOVL C01110 +MOVJ EC01110
SMOVL C01111 +MOVJ EC01111
SMOVL C01112 +MOVJ EC01112
SMOVL C01113 +MOVJ EC01113
SMOVL C01114 +MOVJ EC01114
SMOVL C01115 +MOVJ EC01115
SMOVL C01116 +MOVJ EC01116
SMOVL C01117 +MOVJ EC01117
SMOVL C01118 +MOVJ EC01118
SMOVL C01119 +MOVJ EC01119
SMOVL C01120 +MOVJ EC01120
SMOVL C01121 +MOVJ EC01121
SMOVL C01122 +MOVJ EC01122
SMOVL C01123 +MOVJ EC01123
SMOVL C01124 +MOVJ EC01124
SMOVL C01125 +MOVJ EC01125
SMOVL C01126 +MOVJ EC01126
SMOVL C01127 +MOVJ EC01127
SMOVL C01128 +MOVJ EC01128
SMOVL C01129 +MOVJ EC01129
SMOVL C01130 +MOVJ EC01130
SMOVL C01131 +MOVJ EC01131
SMOVL C01132 +MOVJ EC01132
SMOVL C01133 +MOVJ EC01133
SMOVL C01134 +MOVJ EC01134
SMOVL C01135 +MOVJ EC01135
SMOVL C01136 +MOVJ EC01136
SMOVL C01137 +MOVJ EC01137
SMOVL C01138 +MOVJ EC01138
SMOVL C01139 +MOVJ EC01139
SMOVL C01140 +MOVJ EC01140
SMOVL C01141 +MOVJ EC01141
SMOVL C01142 +MOVJ EC01142
SMOVL C01143 +MOVJ EC01143
SMOVL C01144 +MOVJ EC01144
SMOVL C01145 +MOVJ EC01145
SMOVL C01146 +MOVJ EC01146
SMOVL C01147 +MOVJ EC01147
SMOVL C01148 +MOVJ EC01148
SMOVL C01149 +MOVJ EC01149
SMOVL C01150 +MOVJ EC01150
SMOVL C01151 +MOVJ EC01151
SMOVL C01152 +MOVJ EC01152
SMOVL C01153 +MOVJ EC01153
SMOVL C01154 +MOVJ EC01154
SMOVL C01155 +MOVJ EC01155
SMOVL C01156 +MOVJ EC01156
SMOVL C01157 +MOVJ EC01157
SMOVL C01158 +MOVJ EC01158
SMOVL C01159 +MOVJ EC01159
SMOVL C01160 +MOVJ EC01160
SMOVL C01161 +MOVJ EC01161
SMOVL C01162 +MOVJ EC01162
SMOVL C01163 +MOVJ EC01163
SMOVL C01164 +MOVJ EC01164
SMOVL C01165 +MOVJ EC01165
SMOVL C01166 +MOVJ EC01166
SMOVL C01167 +MOVJ EC01167
SMOVL C01168 +MOVJ EC01168
SMOVL C01169 +MOVJ EC01169
SMOVL C01170 +MOVJ EC01170
SMOVL C01171 +MOVJ EC01171
SMOVL C01172 +MOVJ EC01172
SMOVL C01173 +MOVJ EC01173
SMOVL C01174 +MOVJ EC01174
SMOVL C01175 +MOVJ EC01175
SMOVL C01176 +MOVJ EC01176
SMOVL C01177 +MOVJ EC01177
SMOVL C01178 +MOVJ EC01178
SMOVL C01179 +MOVJ EC01179
SMOVL C01180 +MOVJ EC01180
SMOVL C01181 +MOVJ EC01181
SMOVL C01182 +MOVJ EC01182
SMOVL C01183 +MOVJ EC01183
SMOVL C01184 +MOVJ EC01184
SMOVL C01185 +MOVJ EC01185
SMOVL C01186 +MOVJ EC01186
SMOVL C01187 +MOVJ EC01187
SMOVL C01188 +MOVJ EC01188
SMOVL C01189 +MOVJ EC01189
SMOVL C01190 +MOVJ EC01190
SMOVL C01191 +MOVJ EC01191
SMOVL C01192 +MOVJ EC01192
SMOVL C01193 +MOVJ EC01193
SMOVL C01194 +MOVJ EC01194
SMOVL C01195 +MOVJ EC01195
SMOVL C01196 +MOVJ EC01196
SMOVL C01197 +MOVJ EC01197
SMOVL C01198 +MOVJ EC01198
SMOVL C01199 +MOVJ EC01199
SMOVL C01200 +MOVJ EC01200
SMOVL C01201 +MOVJ EC01201
SMOVL C01202 +MOVJ EC01202
SMOVL C01203 +MOVJ EC01203
SMOVL C01204 +MOVJ EC01204
SMOVL C01205 +MOVJ EC01205
SMOVL C01206 +MOVJ EC01206
SMOVL C01207 +MOVJ EC01207
SMOVL C01208 +MOVJ EC01208
SMOVL C01209 +MOVJ EC01209
SMOVL C01210 +MOVJ EC01210
SMOVL C01211 +MOVJ EC01211
SMOVL C01212 +MOVJ EC01212
SMOVL C01213 +MOVJ EC01213
SMOVL C01214 +MOVJ EC01214
SMOVL C01215 +MOVJ EC01215
SMOVL C01216 +MOVJ EC01216
SMOVL C01217 +MOVJ EC01217
SMOVL C01218 +MOVJ EC01218
SMOVL C01219 +MOVJ EC01219
SMOVL C01220 +MOVJ EC01220
SMOVL C01221 +MOVJ EC01221
SMOVL C01222 +MOVJ EC01222
SMOVL C01223 +MOVJ EC01223
SMOVL C01224 +MOVJ EC01224
SMOVL C01225 +MOVJ EC01225
SMOVL C01226 +MOVJ EC01226
SMOVL C01227 +MOVJ EC01227
SMOVL C01228 +MOVJ EC01228
SMOVL C01229 +MOVJ EC01229
SMOVL C01230 +MOVJ EC01230
SMOVL C01231 +MOVJ EC01231
SMOVL C01232 +MOVJ EC01232
SMOVL C01233 +MOVJ EC01233
SMOVL C01234 +MOVJ EC01234
SMOVL C01235 +MOVJ EC01235
SMOVL C01236 +MOVJ EC01236
SMOVL C01237 +MOVJ EC01237
SMOVL C01238 +MOVJ EC01238
SMOVL C01239 +MOVJ EC01239
SMOVL C01240 +MOVJ EC01240
SMOVL C01241 +MOVJ EC01241
SMOVL C01242 +MOVJ EC01242
SMOVL C01243 +MOVJ EC01243
SMOVL C01244 +MOVJ EC01244
SMOVL C01245 +MOVJ EC01245
SMOVL C01246 +MOVJ EC01246
SMOVL C01247 +MOVJ EC01247
SMOVL C01248 +MOVJ EC01248
SMOVL C01249 +MOVJ EC01249
SMOVL C01250 +MOVJ EC01250
SMOVL C01251 +MOVJ EC01251
SMOVL C01252 +MOVJ EC01252
SMOVL C01253 +MOVJ EC01253
SMOVL C01254 +MOVJ EC01254
SMOVL C01255 +MOVJ EC01255
SMOVL C01256 +MOVJ EC01256
SMOVL C01257 +MOVJ EC01257
SMOVL C01258 +MOVJ EC01258
SMOVL C01259 +MOVJ EC01259
SMOVL C01260 +MOVJ EC01260
SMOVL C01261 +MOVJ EC01261
SMOVL C01262 +MOVJ EC01262
SMOVL C01263 +MOVJ EC01263
SMOVL C01264 +MOVJ EC01264
SMOVL C01265 +MOVJ EC01265
SMOVL C01266 +MOVJ EC01266
SMOVL C01267 +MOVJ EC01267
SMOVL C01268 +MOVJ EC01268
SMOVL C01269 +MOVJ EC01269
SMOVL C01270 +MOVJ EC01270
SMOVL C01271 +MOVJ EC01271
SMOVL C01272 +MOVJ EC01272
SMOVL C01273 +MOVJ EC01273
SMOVL C01274 +MOVJ EC01274
SMOVL C01275 +MOVJ EC01275
SMOVL C01276 +MOVJ EC01276
SMOVL C01277 +MOVJ EC01277
SMOVL C01278 +MOVJ EC01278
SMOVL C01279 +MOVJ EC01279
SMOVL C01280 +MOVJ EC01280
SMOVL C01281 +MOVJ EC01281
SMOVL C01282 +MOVJ EC01282
SMOVL C01283 +MOVJ EC01283
SMOVL C01284 +MOVJ EC01284
SMOVL C01285 +MOVJ EC01285
SMOVL C01286 +MOVJ EC01286
SMOVL C01287 +MOVJ EC01287
SMOVL C01288 +MOVJ EC01288
SMOVL C01289 +MOVJ EC01289
SMOVL C01290 +MOVJ EC01290
SMOVL C01291 +MOVJ EC01291
SMOVL C01292 +MOVJ EC01292
SMOVL C01293 +MOVJ EC01293
SMOVL C01294 +MOVJ EC01294
SMOVL C01295 +MOVJ EC01295
SMOVL C01296 +MOVJ EC01296
SMOVL C01297 +MOVJ EC01297
SMOVL C01298 +MOVJ EC01298
SMOVL C01299 +MOVJ EC01299
SMOVL C01300 +MOVJ EC01300
SMOVL C01301 +MOVJ EC01301
SMOVL C01302 +MOVJ EC01302
SMOVL C01303 +MOVJ EC01303
SMOVL C01304 +MOVJ EC01304
SMOVL C01305 +MOVJ EC01305
SMOVL C01306 +MOVJ EC01306
SMOVL C01307 +MOVJ EC01307
SMOVL C01308 +MOVJ EC01308
SMOVL C01309 +MOVJ EC01309
SMOVL C01310 +MOVJ EC01310
SMOVL C01311 +MOVJ EC01311
SMOVL C01312 +MOVJ EC01312
SMOVL C01313 +MOVJ EC01313
SMOVL C01314 +MOVJ EC01314
SMOVL C01315 +MOVJ EC01315
SMOVL C01316 +MOVJ EC01316
SMOVL C01317 +MOVJ EC01317
SMOVL C01318 +MOVJ EC01318
SMOVL C01319 +MOVJ EC01319
SMOVL C01320 +MOVJ EC01320
SMOVL C01321 +MOVJ EC01321
SMOVL C01322 +MOVJ EC01322
SMOVL C01323 +MOVJ EC01323
SMOVL C01324 +MOVJ EC01324
SMOVL C01325 +MOVJ EC01325
SMOVL C01326 +MOVJ EC01326
SMOVL C01327 +MOVJ EC01327
SMOVL C01328 +MOVJ EC01328
SMOVL C01329 +MOVJ EC01329
SMOVL C01330 +MOVJ EC01330
SMOVL C01331 +MOVJ EC01331
SMOVL C01332 +MOVJ EC01332
SMOVL C01333 +MOVJ EC01333
SMOVL C01334 +MOVJ EC01334
SMOVL C01335 +MOVJ EC01335
SMOVL C01336 +MOVJ EC01336
SMOVL C01337 +MOVJ EC01337
SMOVL C01338 +MOVJ EC01338
SMOVL C01339 +MOVJ EC01339
SMOVL C01340 +MOVJ EC01340
SMOVL C01341 +MOVJ EC01341
SMOVL C01342 +MOVJ EC01342
SMOVL C01343 +MOVJ EC01343
SMOVL C01344 +MOVJ EC01344
SMOVL C01345 +MOVJ EC01345
SMOVL C01346 +MOVJ EC01346
SMOVL C01347 +MOVJ EC01347
SMOVL C01348 +MOVJ EC01348
SMOVL C01349 +MOVJ EC01349
SMOVL C01350 +MOVJ EC01350
SMOVL C01351 +MOVJ EC01351
SMOVL C01352 +MOVJ EC01352
SMOVL C01353 +MOVJ EC01353
SMOVL C01354 +MOVJ EC01354
SMOVL C01355 +MOVJ EC01355
SMOVL C01356 +MOVJ EC01356
SMOVL C01357 +MOVJ EC01357
SMOVL C01358 +MOVJ EC01358
SMOVL C01359 +MOVJ EC01359
SMOVL C01360 +MOVJ EC01360
SMOVL C01361 +MOVJ EC01361
SMOVL C01362 +MOVJ EC01362
SMOVL C01363 +MOVJ EC01363
SMOVL C01364 +MOVJ EC01364
SMOVL C01365 +MOVJ EC01365
SMOVL C01366 +MOVJ EC01366
SMOVL C01367 +MOVJ EC01367
SMOVL C01368 +MOVJ EC01368
SMOVL C01369 +MOVJ EC01369
SMOVL C01370 +MOVJ EC01370
SMOVL C01371 +MOVJ EC01371
SMOVL C01372 +MOVJ EC01372
SMOVL C01373 +MOVJ EC01373
SMOVL C01374 +MOVJ EC01374
SMOVL C01375 +MOVJ EC01375
SMOVL C01376 +MOVJ EC01376
SMOVL C01377 +MOVJ EC01377
SMOVL C01378 +MOVJ EC01378
SMOVL C01379 +MOVJ EC01379
SMOVL C01380 +MOVJ EC01380
SMOVL C01381 +MOVJ EC01381
SMOVL C01382 +MOVJ EC01382
SMOVL C01383 +MOVJ EC01383
SMOVL C01384 +MOVJ EC01384
SMOVL C01385 +MOVJ EC01385
SMOVL C01386 +MOVJ EC01386
SMOVL C01387 +MOVJ EC01387
SMOVL C01388 +MOVJ EC01388
SMOVL C01389 +MOVJ EC01389
SMOVL C01390 +MOVJ EC01390
SMOVL C01391 +MOVJ EC01391
SMOVL C01392 +MOVJ EC01392
SMOVL C01393 +MOVJ EC01393
SMOVL C01394 +MOVJ EC01394
SMOVL C01395 +MOVJ EC01395
SMOVL C01396 +MOVJ EC01396
SMOVL C01397 +MOVJ EC01397
SMOVL C01398 +MOVJ EC01398
SMOVL C01399 +MOVJ EC01399
SMOVL C01400 +MOVJ EC01400
SMOVL C01401 +MOVJ EC01401
SMOVL C01402 +MOVJ EC01402
SMOVL C01403 +MOVJ EC01403
SMOVL C01404 +MOVJ EC01404
SMOVL C01405 +MOVJ EC01405
SMOVL C01406 +MOVJ EC01406
SMOVL C01407 +MOVJ EC01407
SMOVL C01408 +MOVJ EC01408
SMOVL C01409 +MOVJ EC01409
SMOVL C01410 +MOVJ EC01410
SMOVL C01411 +MOVJ EC01411
SMOVL C01412 +MOVJ EC01412
SMOVL C01413 +MOVJ EC01413
SMOVL C01414 +MOVJ EC01414
SMOVL C01415 +MOVJ EC01415
SMOVL C01416 +MOVJ EC01416
SMOVL C01417 +MOVJ EC01417
SMOVL C01418 +MOVJ EC01418
SMOVL C01419 +MOVJ EC01419
SMOVL C01420 +MOVJ EC01420
SMOVL C01421 +MOVJ EC01421
SMOVL C01422 +MOVJ EC01422
SMOVL C01423 +MOVJ EC01423
SMOVL C01424 +MOVJ EC01424
SMOVL C01425 +MOVJ EC01425
SMOVL C01426 +MOVJ EC01426
SMOVL C01427 +MOVJ EC01427
SMOVL C01428 +MOVJ EC01428
SMOVL C01429 +MOVJ EC01429
SMOVL C01430 +MOVJ EC01430
SMOVL C01431 +MOVJ EC01431
SMOVL C01432 +MOVJ EC01432
SMOVL C01433 +MOVJ EC01433
SMOVL C01434 +MOVJ EC01434
SMOVL C01435 +MOVJ EC01435
SMOVL C01436 +MOVJ EC01436
SMOVL C01437 +MOVJ EC01437
SMOVL C01438 +MOVJ EC01438
SMOVL C01439 +MOVJ EC01439
SMOVL C01440 +MOVJ EC01440
SMOVL C01441 +MOVJ EC01441
SMOVL C01442 +MOVJ EC01442
SMOVL C01443 +MOVJ EC01443
SMOVL C01444 +MOVJ EC01444
SMOVL C01445 +MOVJ EC01445
SMOVL C01446 +MOVJ EC01446
SMOVL C01447 +MOVJ EC01447
SMOVL C01448 +MOVJ EC01448
SMOVL C01449 +MOVJ EC01449
SMOVL C01450 +MOVJ EC01450
SMOVL C01451 +MOVJ EC01451
SMOVL C01452 +MOVJ EC01452
SMOVL C01453 +MOVJ EC01453
SMOVL C01454 +MOVJ EC01454
SMOVL C01455 +MOVJ EC01455
SMOVL C01456 +MOVJ EC01456
SMOVL C01457 +MOVJ EC01457
SMOVL C01458 +MOVJ EC01458
SMOVL C01459 +MOVJ EC01459
SMOVL C01460 +MOVJ EC01460
SMOVL C01461 +MOVJ EC01461
SMOVL C01462 +MOVJ EC01462
SMOVL C01463 +MOVJ EC01463
SMOVL C01464 +MOVJ EC01464
SMOVL C01465 +MOVJ EC01465
SMOVL C01466 +MOVJ EC01466
SMOVL C01467 +MOVJ EC01467
SMOVL C01468 +MOVJ EC01468
SMOVL C01469 +MOVJ EC01469
SMOVL C01470 +MOVJ EC01470
SMOVL C01471 +MOVJ EC01471
SMOVL C01472 +MOVJ EC01472
SMOVL C01473 +MOVJ EC01473
SMOVL C01474 +MOVJ EC01474
SMOVL C01475 +MOVJ EC01475
SMOVL C01476 +MOVJ EC01476
SMOVL C01477 +MOVJ EC01477
SMOVL C01478 +MOVJ EC01478
SMOVL C01479 +MOVJ EC01479
SMOVL C01480 +MOVJ EC01480
SMOVL C01481 +MOVJ EC01481
SMOVL C01482 +MOVJ EC01482
SMOVL C01483 +MOVJ EC01483
SMOVL C01484 +MOVJ EC01484
SMOVL C01485 +MOVJ EC01485
SMOVL C01486 +MOVJ EC01486
SMOVL C01487 +MOVJ EC01487
SMOVL C01488 +MOVJ EC01488
SMOVL C01489 +MOVJ EC01489
SMOVL C01490 +MOVJ EC01490
SMOVL C01491 +MOVJ EC01491
SMOVL C01492 +MOVJ EC01492
SMOVL C01493 +MOVJ EC01493
SMOVL C01494 +MOVJ EC01494
SMOVL C01495 +MOVJ EC01495
SMOVL C01496 +MOVJ EC01496
SMOVL C01497 +MOVJ EC01497
SMOVL C01498 +MOVJ EC01498
SMOVL C01499 +MOVJ EC01499
SMOVL C01500 +MOVJ EC01500
SMOVL C01501 +MOVJ EC01501
SMOVL C01502 +MOVJ EC01502
SMOVL C01503 +MOVJ EC01503
SMOVL C01504 +MOVJ EC01504
SMOVL C01505 +MOVJ EC01505
SMOVL C01506 +MOVJ EC01506
SMOVL C01507 +MOVJ EC01507
SMOVL C01508 +MOVJ EC01508
SMOVL C01509 +MOVJ EC01509
SMOVL C01510 +MOVJ EC01510
SMOVL C01511 +MOVJ EC01511
SMOVL C01512 +MOVJ EC01512
SMOVL C01513 +MOVJ EC01513
SMOVL C01514 +MOVJ EC01514
SMOVL C01515 +MOVJ EC01515
SMOVL C01516 +MOVJ EC01516
SMOVL C01517 +MOVJ EC01517
SMOVL C01518 +MOVJ EC01518
SMOVL C01519 +MOVJ EC01519
SMOVL C01520 +MOVJ EC01520
SMOVL C01521 +MOVJ EC01521
SMOVL C01522 +MOVJ EC01522
SMOVL C01523 +MOVJ EC01523
SMOVL C01524 +MOVJ EC01524
SMOVL C01525 +MOVJ EC01525
SMOVL C01526 +MOVJ EC01526
SMOVL C01527 +MOVJ EC01527
SMOVL C01528 +MOVJ EC01528
SMOVL C01529 +MOVJ EC01529
SMOVL C01530 +MOVJ EC01530
SMOVL C01531 +MOVJ EC01531
SMOVL C01532 +MOVJ EC01532
SMOVL C01533 +MOVJ EC01533
SMOVL C01534 +MOVJ EC01534
SMOVL C01535 +MOVJ EC01535
SMOVL C01536 +MOVJ EC01536
SMOVL C01537 +MOVJ EC01537
SMOVL C01538 +MOVJ EC01538
SMOVL C01539 +MOVJ EC01539
SMOVL C01540 +MOVJ EC01540
SMOVL C01541 +MOVJ EC01541
SMOVL C01542 +MOVJ EC01542
SMOVL C01543 +MOVJ EC01543
SMOVL C01544 +MOVJ EC01544
SMOVL C01545 +MOVJ EC01545
SMOVL C01546 +MOVJ EC01546
SMOVL C01547 +MOVJ EC01547
SMOVL C01548 +MOVJ EC01548
SMOVL C01549 +MOVJ EC01549
SMOVL C01550 +MOVJ EC01550
SMOVL C01551 +MOVJ EC01551
SMOVL C01552 +MOVJ EC01552
SMOVL C01553 +MOVJ EC01553
SMOVL C01554 +MOVJ EC01554
SMOVL C01555 +MOVJ EC01555
SMOVL C01556 +MOVJ EC01556
SMOVL C01557 +MOVJ EC01557
SMOVL C01558 +MOVJ EC01558
SMOVL C01559 +MOVJ EC01559
SMOVL C01560 +MOVJ EC01560
SMOVL C01561 +MOVJ EC01561
SMOVL C01562 +MOVJ EC01562
SMOVL C01563 +MOVJ EC01563
SMOVL C01564 +MOVJ EC01564
SMOVL C01565 +MOVJ EC01565
SMOVL C01566 +MOVJ EC01566
SMOVL C01567 +MOVJ EC01567
SMOVL C01568 +MOVJ EC01568
SMOVL C01569 +MOVJ EC01569
SMOVL C01570 +MOVJ EC01570
SMOVL C01571 +MOVJ EC01571
SMOVL C01572 +MOVJ EC01572
SMOVL C01573 +MOVJ EC01573
SMOVL C01574 +MOVJ EC01574
SMOVL C01575 +MOVJ EC01575
SMOVL C01576 +MOVJ EC01576
SMOVL C01577 +MOVJ EC01577
SMOVL C01578 +MOVJ EC01578
SMOVL C01579 +MOVJ EC01579
SMOVL C01580 +MOVJ EC01580
SMOVL C01581 +MOVJ EC01581
SMOVL C01582 +MOVJ EC01582
SMOVL C01583 +MOVJ EC01583
SMOVL C01584 +MOVJ EC01584
SMOVL C01585 +MOVJ EC01585
SMOVL C01586 +MOVJ EC01586
SMOVL C01587 +MOVJ EC01587
SMOVL C01588 +MOVJ EC01588
SMOVL C01589 +MOVJ EC01589
SMOVL C01590 +MOVJ EC01590
SMOVL C01591 +MOVJ EC01591
SMOVL C01592 +MOVJ EC01592
SMOVL C01593 +MOVJ EC01593
SMOVL C01594 +MOVJ EC01594
SMOVL C01595 +MOVJ EC01595
SMOVL C01596 +MOVJ EC01596
SMOVL C01597 +MOVJ EC01597
SMOVL C01598 +MOVJ EC01598
SMOVL C01599 +MOVJ EC01599
SMOVL C01600 +MOVJ EC01600
SMOVL C01601 +MOVJ EC01601
SMOVL C01602 +MOVJ EC01602
SMOVL C01603 +MOVJ EC01603
SMOVL C01604 +MOVJ EC01604
SMOVL C01605 +MOVJ EC01605
SMOVL C01606 +MOVJ EC01606
SMOVL C01607 +MOVJ EC01607
SMOVL C01608 +MOVJ EC01608
SMOVL C01609 +MOVJ EC01609
SMOVL C01610 +MOVJ EC01610
SMOVL C01611 +MOVJ EC01611
SMOVL C01612 +MOVJ EC01612
SMOVL C01613 +MOVJ EC01613
SMOVL C01614 +MOVJ EC01614
SMOVL C01615 +MOVJ EC01615
SMOVL C01616 +MOVJ EC01616
SMOVL C01617 +MOVJ EC01617
SMOVL C01618 +MOVJ EC01618
SMOVL C01619 +MOVJ EC01619
SMOVL C01620 +MOVJ EC01620
SMOVL C01621 +MOVJ EC01621
SMOVL C01622 +MOVJ EC01622
SMOVL C01623 +MOVJ EC01623
SMOVL C01624 +MOVJ EC01624
SMOVL C01625 +MOVJ EC01625
SMOVL C01626 +MOVJ EC01626
SMOVL C01627 +MOVJ EC01627
SMOVL C01628 +MOVJ EC01628
SMOVL C01629 +MOVJ EC01629
SMOVL C01630 +MOVJ EC01630
SMOVL C01631 +MOVJ EC01631
SMOVL C01632 +MOVJ EC01632
SMOVL C01633 +MOVJ EC01633
SMOVL C01634 +MOVJ EC01634
SMOVL C01635 +MOVJ EC01635
SMOVL C01636 +MOVJ EC01636
SMOVL C01637 +MOVJ EC01637
SMOVL C01638 +MOVJ EC01638
SMOVL C01639 +MOVJ EC01639
SMOVL C01640 +MOVJ EC01640
SMOVL C01641 +MOVJ EC01641
SMOVL C01642 +MOVJ EC01642
SMOVL C01643 +MOVJ EC01643
SMOVL C01644 +MOVJ EC01644
SMOVL C01645 +MOVJ EC01645
SMOVL C01646 +MOVJ EC01646
SMOVL C01647 +MOVJ EC01647
SMOVL C01648 +MOVJ EC01648
SMOVL C01649 +MOVJ EC01649
SMOVL C01650 +MOVJ EC01650
SMOVL C01651 +MOVJ EC01651
SMOVL C01652 +MOVJ EC01652
SMOVL C01653 +MOVJ EC01653
SMOVL C01654 +MOVJ EC01654
SMOVL C01655 +MOVJ EC01655
SMOVL C01656 +MOVJ EC01656
SMOVL C01657 +MOVJ EC01657
SMOVL C01658 +MOVJ EC01658
SMOVL C01659 +MOVJ EC01659
SMOVL C01660 +MOVJ EC01660
SMOVL C01661 +MOVJ EC01661
SMOVL C01662 +MOVJ EC01662
SMOVL C01663 +MOVJ EC01663
SMOVL C01664 +MOVJ EC01664
SMOVL C01665 +MOVJ EC01665
SMOVL C01666 +MOVJ EC01666
SMOVL C01667 +MOVJ EC01667
SMOVL C01668 +MOVJ EC01668
SMOVL C01669 +MOVJ EC01669
SMOVL C01670 +MOVJ EC01670
SMOVL C01671 +MOVJ EC01671
SMOVL C01672 +MOVJ EC01672
SMOVL C01673 +MOVJ EC01673
SMOVL C01674 +MOVJ EC01674
SMOVL C01675 +MOVJ EC01675
SMOVL C01676 +MOVJ EC01676
